# B&R Automation Studio project EFI (part 15)

#### Motors.st
```iecst
ACTION dataToMotors:
	rJogSpeedSetPoint:=data.parameters.JogSpeed;

	//Drive Unit data Managment
	MotorDriveUnit.TransmissionData := data.parameters.DriveUnit;

	MotorDriveUnit.HomePositionDesired:=data.Motor[iIndexIclaMotor].rHomePosition;;
	MotorDriveUnit.Calculation:=CALC_HOMEPOS_PULSES;
	MotorDriveUnit();

	MotorDriveUnit.SpeedDesired:=data.parameters.Speed;
	MotorDriveUnit.Calculation:=CALC_SPEED_PULSES;
	MotorDriveUnit();

	MotorDriveUnit.JogSpeedDesired:=rJogSpeedSetPoint;
	MotorDriveUnit.Calculation:=CALC_JOGSPEED_PULSES;
	MotorDriveUnit();

	MotorDriveUnit.AccelerationDesired:=data.parameters.Acceleration;
	MotorDriveUnit.Calculation:=CALC_ACC_PULSES;
	MotorDriveUnit();

	AssignDataToMotors;
END_ACTION

ACTION AssignDataToMotors:

	//Position
	//IclaMotors[iIndexIclaMotor].Parameter.MoveAbsolute.Position := REAL_TO_DINT(MotorDriveUnit.pulsesPositionDesired);

	//Speed
	IclaMotors[iIndexIclaMotor].Parameter.MoveAbsolute.Velocity := REAL_TO_UINT(MotorDriveUnit.pulsesSpeedDesired);

	//Jog Speed
	IclaMotors[iIndexIclaMotor].Parameter.Jog.VeloSlow 			:= REAL_TO_UINT(MotorDriveUnit.pulsesJogSpeedDesired);
	IclaMotors[iIndexIclaMotor].Command.JogFastSpeed 			:= FALSE;

	//Acceleration
	IclaMotors[iIndexIclaMotor].Parameter.iAcceleration 		:= REAL_TO_UINT(MotorDriveUnit.pulsesAccelerationDesired);

	//Home
	IclaMotors[iIndexIclaMotor].Parameter.Home.Position 		:= REAL_TO_DINT(MotorDriveUnit.pulsesHomePositionDesired);

	//Reset
	IclaMotors[iIndexIclaMotor].Command.Reset 					:= 	data.commands.xResetMotor OR (data.commands.xErrorRst AND
																	IclaMotors[iIndexIclaMotor].Status.IclaStatus <> AXISILE_MOVE_ABSOLUTE AND
																	IclaMotors[iIndexIclaMotor].Status.IclaStatus <> AXISILE_JOG AND
																	IclaMotors[iIndexIclaMotor].Status.IclaStatus <> AXISILE_HOMING);

END_ACTION

ACTION dataFromMotors:

	xAnyManualMovement:= (IclaMotors[iIndexIclaMotor].Status.IclaStatus = AXISILE_JOG);

	MotorDriveUnit.pulsesDevice 	:= DINT_TO_REAL(IclaMotors[iIndexIclaMotor].Status.iActualPosition);
	MotorDriveUnit.PulsesSpeedDevice:=IclaMotors[iIndexIclaMotor].Status.iActualVelocity;

	// Conversions
	MotorDriveUnit.Calculation:= CALC_POS_MM;
	MotorDriveUnit();
	rPositionMotorMm := data.Motor[iIndexIclaMotor].iDirection * MotorDriveUnit.PositionDevice;

	data.Motor[iIndexIclaMotor].rPositionMotor := rPositionMotorMm;
	data.Motor[iIndexIclaMotor].rMetalStrapPos := ABS(rPositionMotorMm)*2 + gEdgeHoldDown.Hw.rMinWidthAdjustment;

	MotorDriveUnit.Calculation:= CALC_SPEED_MM;
	MotorDriveUnit();

END_ACTION
```

- Program Logical/ExtPack/_Transport/PairedIclaMotors/PairedIclaMotorsSim/PairedIclaMotorsSim_v1/PairedIclaMotorsSim (IEC) (no source held here)

### Program Logical/ExtPack/_Transport/PairedIclaMotors/PairedIclaMotorsSim/PairedIclaMotorsSim_v1/InitPairedIclaMotorsSim (IEC)

#### InitPairedIclaMotorsSim.st
```iecst
PROGRAM _CYCLIC
	iPairedIclaMotorSimIndex := 1;
END_PROGRAM
```

### Program Logical/ExtPack/_Transport/TransVacuumCtrl/TransVacuumCtrl_v1/TransVacuumCtrl (IEC)

#### TransVacuumCtrl.var
```iecst
VAR
	dataVacc : REFERENCE TO TransVacuum_typ;
	AlarmsSummaryReseted : stEFI_AlarmSummary;
	AlarmsReseted : TransVacuumAlarms_typ;
	CommandsReseted : TransVacuumCommands_typ;
	Blower : REFERENCE TO AxisP66_typ;
	BlowersWatch : ARRAY[1..MAX_LAST_MOTOR_BLOWER] OF AxisP66_typ;
	ConditionStart_copy : BOOL; (*Storing all previous data*)
	ConditionStart : BOOL; (*Storing all previous data*)
	ConditionsStart_copy : ARRAY[1..MAX_LAST_MOTOR_BLOWER] OF BOOL; (*Storing all previous data*)
	rVacPressure : REAL; (*Pressure measured by the sensor*)
	rVacPressurePerc : REAL; (*Pressure measured by the sensor in % of MaxSystemVacuum*)
	xEnablePID : BOOL;
	xUpdatePID : BOOL;
	fbPIDPressure : MTBasicsPID;
	pidParPressure : MTPIDParametersType;
	StatusCtrl : TransVacuumStatusCtrl;
	xRunBlowerAuto : BOOL;
	xRunOutOfProduction : BOOL;
	xRunBlowerMan : BOOL;
	iReasonStop : UDINT;
	iReasonCritical : UDINT;
	iReasonSound : UDINT;
	arxAlrVacuumSensor : AutoResetSound;
	arxAlrComsBlower : AutoResetSound;
	arxAlrDriveBlowerError : AutoResetSound;
	stEventLog : EventLog_typ;
	tonJunctionAlarm : TON;
	arxAlrJointSystemPressure : AutoResetSound;
	arxAlrBlowerCB : AutoResetSound;
	uiIndex : USINT;
	StatusCtrl_copy : TransVacuumStatusCtrl;
	FLP_PresFilterPasLow : MTFilterLowPass;
	TON_StopBlowersDly : TON; (*Delay to filter fast pause-start transcition*)
	xLabStartedBlowers : BOOL; (*Blowers started for first time un the laboratory mode*)
	xAllBlowersAtSpeed : BOOL;
	xAllBlowersRunning : BOOL;
	BlowerDirection : MotorDirection_enum;
	BlowerDirectionsWatch : ARRAY[1..MAX_LAST_MOTOR_BLOWER] OF MotorDirection_enum;
	tonBlowerNotRunning : ARRAY[1..MAX_LAST_MOTOR_BLOWER] OF TON;
	iReasonOutOfProduction : UINT;
	iReasonRunAuto : USINT;
	xDisableBlower : ARRAY[1..MAX_LAST_MOTOR_BLOWER] OF BOOL;
	xAllBlowerDisabled : BOOL;
	tonBlowersRunning : TON;
	xProductionOrJamRecovery : BOOL;
	tpEvEvacuateInk : TP;
	tofNotStartAfterEStop : TOF;
	iAnyWarning : USINT;
	tonCheckAlarms : TON;
	xEnteringPowerOn : BOOL;
END_VAR
```

#### Alarms.st
```iecst
ACTION Alarms:

	IF dataVacc.Inputs.xPressureSensorError AND (xProductionOrJamRecovery OR xRunOutOfProduction) THEN
		dataVacc.Alarms.xAlrVacuumSensor := TRUE;
	END_IF

	IF dataVacc.Parameters.Hw.xSystemWithJoints THEN
		tonJunctionAlarm.IN:= NOT dataVacc.Inputs.xJointSystemPressure AND StatusCtrl<>TRANSVAC_OFF;
		tonJunctionAlarm.PT:= T#500ms;
		tonJunctionAlarm();
	END_IF

	IF tonJunctionAlarm.Q  THEN
		dataVacc.Alarms.xAlrJointSystemPressure := TRUE;
	END_IF

	IF dataVacc.Inputs.xBlowersAnyCB THEN
		dataVacc.Alarms.xAlrBlowersAnyCB := TRUE;
	END_IF

	//////////////////////////////////////////////////////////////
	// ALARMS SUMMARY    ALARMS SUMMARY    ALARMS SUMMARY

	iReasonStop.0 := dataVacc.Alarms.xAlrVacuumSensor; //To enable go to ByPass with a sensor error
	iReasonStop.1 := dataVacc.Alarms.xAlrComsBlower;
	iReasonStop.2 := dataVacc.Alarms.xAlrDriveBlowerError;
	iReasonStop.3 := dataVacc.Alarms.xAlrOvertorque;
	iReasonStop.4 := dataVacc.Alarms.xAlrJointSystemPressure AND NOT dataVacc.Parameters.AutoMode.xBypass;
	iReasonStop.5 := dataVacc.Alarms.xAlrBlowersAnyCB;
	iReasonStop.6 := dataVacc.Alarms.xAlrBlowerCB[1];
	iReasonStop.7 := dataVacc.Alarms.xAlrBlowerCB[2];
	iReasonStop.8 := dataVacc.Alarms.xAlrBlowerNotRunning[1];
	iReasonStop.9 := dataVacc.Alarms.xAlrBlowerNotRunning[2];

	IF (dataVacc.Parameters.AutoMode.xProduction OR (dataVacc.parSw.xActiveOutOfProduction AND (dataVacc.Parameters.AutoMode.xLaboratory OR dataVacc.Parameters.AutoMode.xBypass))) THEN
		dataVacc.AlSummary.xAlarmStop:=	iReasonStop > 0;
		IF EDGEPOS(dataVacc.AlSummary.xAlarmStop) THEN
			dataVacc.AlSummary.iReasonStop[0] := iReasonStop;
			LogStopAlarm;
		ELSIF EDGEPOS(NOT dataVacc.Parameters.AutoMode.xStop AND NOT dataVacc.AlSummary.xAlarmStop) THEN
			dataVacc.AlSummary.iReasonStop[0] := 0;
		END_IF
	END_IF

	dataVacc.AlSummary.xAlarmCritical := iReasonCritical > 0;
	IF EDGEPOS(dataVacc.AlSummary.xAlarmCritical) THEN
		dataVacc.AlSummary.iReasonCritical := iReasonCritical;
	ELSIF EDGEPOS(dataVacc.Parameters.Mode.xAuto AND NOT dataVacc.AlSummary.xAlarmCritical) THEN
		dataVacc.AlSummary.iReasonCritical := 0;
	END_IF

	//Warning
	// It is just used for drive alarms
	iAnyWarning.0 := dataVacc.Alarms.xAlrBlowerNotRunning[1];
	iAnyWarning.1 := dataVacc.Alarms.xAlrBlowerNotRunning[2];
	dataVacc.AlSummary.xAnyWarning:= iAnyWarning > 0;

	IF EDGEPOS(dataVacc.AlSummary.xAnyWarning) THEN
		dataVacc.AlSummary.iReasonWarning := iAnyWarning;
		//LogWarningAlarm;
	ELSIF EDGENEG(dataVacc.AlSummary.xAnyWarning) THEN
		dataVacc.AlSummary.iReasonWarning := 0;
	END_IF

	// Reseteable alarms
	arxAlrVacuumSensor.xAlarm   := dataVacc.Alarms.xAlrVacuumSensor;
	arxAlrVacuumSensor.xSilence := dataVacc.Commands.xMute;
	arxAlrVacuumSensor();

	arxAlrComsBlower.xAlarm   := dataVacc.Alarms.xAlrComsBlower;
	arxAlrComsBlower.xSilence := dataVacc.Commands.xMute;
	arxAlrComsBlower();

	arxAlrDriveBlowerError.xAlarm   := dataVacc.Alarms.xAlrDriveBlowerError;
	arxAlrDriveBlowerError.xSilence := dataVacc.Commands.xMute;
	arxAlrDriveBlowerError();

	arxAlrJointSystemPressure.xAlarm   := dataVacc.Alarms.xAlrJointSystemPressure;
	arxAlrJointSystemPressure.xSilence := dataVacc.Commands.xMute;
	arxAlrJointSystemPressure();

	arxAlrBlowerCB.xAlarm	:=	dataVacc.Alarms.xAlrBlowersAnyCB OR
								dataVacc.Alarms.xAlrBlowerCB[1] OR
								dataVacc.Alarms.xAlrBlowerCB[2];

	arxAlrBlowerCB.xSilence	:= dataVacc.Commands.xMute;
	arxAlrBlowerCB();

	iReasonSound.0 := arxAlrVacuumSensor.xAlarmSound;
	iReasonSound.1 := arxAlrComsBlower.xAlarmSound;
	iReasonSound.2 := arxAlrDriveBlowerError.xAlarmSound;
	iReasonSound.3 := arxAlrJointSystemPressure.xAlarmSound;
	iReasonSound.4 := arxAlrBlowerCB.xAlarmSound;
	dataVacc.AlSummary.xAlarmSound:= iReasonSound > 0;

	// Mute sound in belt alarms
	IF dataVacc.Commands.xMute OR dataVacc.Commands.xReset THEN
		dataVacc.AlSummary.xAlarmSound:= FALSE;
	END_IF

END_ACTION

ACTION ResetAlarms:
	dataVacc.Alarms := AlarmsReseted;
	dataVacc.AlSummary := AlarmsSummaryReseted;
END_ACTION
```

### TransVacuumSim.var
```iecst
VAR
	iTransVacummSimIndex : USINT;
END_VAR
```

### Program Logical/ExtPack/_Transport/TransVacuumCtrl/TransVacuumSim/TransVacuumSim_v1/InitTransVacuumSim

#### Cyclic.st
```iecst
PROGRAM _CYCLIC
	(* Insert code here *)
	iTransVacummSimIndex := 1;

END_PROGRAM
```

### Program Logical/ExtPack/_Transport/TransVacuumCtrl/TransVacuumSim/TransVacuumSim_v1/TransVacuumSim (IEC)

#### TransVacuumSim.var - Local variables
```iecst
VAR
	transVacc : REFERENCE TO TransVacuum_typ;
	pressureSim : SimAnalogProcess;
	rAParam : REAL := -0.13;
	rBParam : REAL := -0.005;
	tofNoVacc : TOF;
END_VAR
```

### Program Logical/ExtPack/BlockCtrl/BlockCtrl_v1/BlockCtrl (IEC) - Block program

#### BlockParameters.st
```iecst
ACTION BlockParameters:

	//Cleaning offset limits.(antes en securities)
	Block.parSw.rOffsetCleanMtrAdjust	:= LIMIT(Block.parameters.Motor.rMinCleanOffsetTech, Block.parSw.rOffsetCleanMtrAdjust, Block.parameters.Motor.rMaxCleanOffsetTech);
	Block.parSw.rOffsetCleanMtrOperatr := LIMIT(-1, Block.parSw.rOffsetCleanMtrOperatr, 1);

	// Clean offset
	rOffseCleanMtr:=Block.parSw.rOffsetCleanMtrAdjust+Block.parSw.rOffsetCleanMtrOperatr;

	//Minimum position of the Motor to allow moving the Icla in Manual mode
	rSafeBarPosToCarrier := Block.parameters.Motor.rSafePositionCleanCarrier; //Block.parameters.Motor.rCleanPosition + rOffseCleanMtr;

	// rWaterSpurtPosition always has to be higher than rCleanPosition
	IF Block.parameters.Motor.rWaterSpurtPosition <= Block.parameters.Motor.rCleanPosition + 0.5 THEN
		Block.parameters.Motor.rWaterSpurtPosition := Block.parameters.Motor.rCleanPosition + 0.5;
	END_IF

	// Print motor offset
	IF NOT Block.parameters.xMotorOffsetAllowed THEN
		Block.parSw.rOffsetPrintMotor := 0;
	ELSE
		Block.parSw.rOffsetPrintMotor := MAX(Block.parSw.rOffsetPrintMotor,GC_MIN_OFFSET_BLOCK);
	END_IF

	// Clean motor speed limits
	Block.parameters.Icla.iCleanMotorSpeedFwd:= LIMIT(Block.parameters.Icla.iMinSpeedCleanMotorFwd,
														Block.parameters.Icla.iCleanMotorSpeedFwd,
														Block.parameters.Icla.iMaxSpeedCleanMotorFwd);

	Block.parameters.Icla.iCleanMotorSpeedBwd:= LIMIT(Block.parameters.Icla.iMinSpeedCleanMotorBwd,
														Block.parameters.Icla.iCleanMotorSpeedBwd,
														Block.parameters.Icla.iMaxSpeedCleanMotorBwd);

	//Assign the direction of the vertical motor
	IF Block.parameters.Motor.VerticalDirection=MOTOR_NEGATIVE THEN
		AxisBK.Parameter.Direction:=MOTOR_NEGATIVE_AXIS;
	ELSE
		AxisBK.Parameter.Direction:=MOTOR_POSITIVE_AXIS;
	END_IF

	Block.parameters.Inks.iMaxMachinePrintBars := MIN(Block.parameters.Inks.iMaxMachinePrintBars, MAX_LAST_INK);

END_ACTION
```

#### AlarmSound.st - Assign sound to alarms
```iecst
ACTION AlarmSound:

	//////////////////////////////
	// BLOCK SOUNDS
	//////////////////////////////

	// Block sounds while is homing
	// Sound generation for homing process
	// Sound generation: manual movements
	xAnyManualMov	:=	Block.Status.Motor.xBarsHoming OR
						AxisBK.Command.Jog.ContinuousPos OR
						AxisBK.Command.Jog.ContinuousNeg OR
						IclaBK.Command.JogForward OR
						IclaBK.Command.JogBackward;

	// Reseteable alarms. Reset is input in the ars function
	// Alarms reseteable sound management.
	ars_AlrStop.xAlarm:= Block.AlSummary.xAlarmStop;
	ars_AlrStop.xSilence:= Block.commands.xMute;
	ars_AlrStop();

	ars_AlrCritical.xAlarm:= Block.AlSummary.xAlarmCritical;
	ars_AlrCritical.xSilence:= Block.commands.xMute;
	ars_AlrCritical();

	ars_AlrWarning.xAlarm:= Block.AlSummary.xAnyWarning;
	ars_AlrWarning.xSilence:= Block.commands.xMute;
	ars_AlrWarning();

	//reasonSound.0 := ars_AlrWarning.xAlarmSound;  //[RGP] I think warnings shouldnt sound
	reasonSound.1 := ars_AlrStop.xAlarmSound;
	reasonSound.2 := ars_AlrCritical.xAlarmSound;
	reasonSound.3 := (xAnyManualMov AND gPLC.xBlk_200ms);

	Block.AlSummary.xAlarmSound := reasonSound>0;

END_ACTION
```

#### AlarmsSummary.st - Alarms summary
```iecst
ACTION AlarmsSummary:

	// Stop Alarms. The machine goes to Automatic-Stop.
	iReasonStop.0 := Block.Al.xAlrCleanMtrNoRef;
	iReasonStop.1 := Block.Al.xAlAirVenturi AND Block.Status.PositionState = BLOCKP_CLEANING;
	iReasonStop.2 := Block.Al.xAnyVerticalDriveAlarm;
	iReasonStop.3 := Block.Al.xAlrBarMtrNoRef;
	iReasonStop.4 := Block.Al.xSiUnitPowerOff;
	iReasonStop.5 := Block.Al.xAlrComSiUnit;
	iReasonStop.6 := Block.Al.xAlrComBarMtr;
	iReasonStop.7 := Block.Al.xAlrCleanMotor;
	iReasonStop.8 := Block.Al.xAlrComCleanMtr;
	iReasonStop.9 := Block.Al.xAlrEnabCleanMtrDiffLvL;
	iReasonStop.10 := Block.Al.xAlrIncoherPositCleanMtr;
	iReasonStop.11 := Block.Al.xAlCleanInterrupt AND Block.commands.AutoMode.xProdORLab;
	iReasonStop.12 := (Block.Al.xAlrTraySensor OR Block.Al.xAlrCleanSensor) AND Block.commands.AutoMode.xProdORLab;
	iReasonStop.13 := Block.Al.xNoActionDangerCollision;
	iReasonStop.14 := Block.Al.xAlrControllerNotReady;
	iReasonStop.15 := Block.Al.xAlrOverTorque;

	Block.AlSummary.xAlarmStop:= iReasonStop > 0;
	IF EDGEPOS(Block.AlSummary.xAlarmStop) THEN
		Block.AlSummary.iReasonStop[0] := iReasonStop;
		LogStopAlarm;
	ELSIF EDGEPOS(NOT Block.commands.AutoMode.xStop AND NOT Block.AlSummary.xAlarmStop) THEN
		Block.AlSummary.iReasonStop[0] := 0;
	END_IF

	// Out of Automatic Alarms. The machine goes to Standby mode.
	iReasonCritical.0 := (Block.Al.xAlrSafetySystemInBlock AND Block.Status.xEnabledMovements);
	iReasonCritical.1 := Block.Al.xAlrDif;
	iReasonCritical.2 := Block.Al.xAlrDriveProtection;
	Block.AlSummary.xAlarmCritical:= iReasonCritical > 0;

	//Register the reason of the Critical Alarm
	IF Block.commands.Mode.xAuto AND EDGEPOS(Block.AlSummary.xAlarmCritical) THEN
		Block.AlSummary.iReasonCritical := iReasonCritical;
		LogCriticalAlarm;
	ELSIF EDGEPOS(Block.commands.Mode.xAuto AND NOT Block.AlSummary.xAlarmCritical) THEN
		Block.AlSummary.iReasonCritical := 0;
	END_IF

	// Any alarm
	Block.AlSummary.xAnyAlarm:= Block.AlSummary.xAlarmStop OR Block.AlSummary.xAlarmCritical;

	// Warning alarms (used in AlarmaAvisoExterno)
	iReasonAnyWarning.0 := Block.Al.xAlrNoTrayInServoNoHomed;
	iReasonAnyWarning.1 := Block.Al.xModuleTemp01;
	iReasonAnyWarning.2 := Block.Al.xModuleTemp02;
	iReasonAnyWarning.3 := Block.Al.xModuleTemp03;
	iReasonAnyWarning.4 := Block.Al.xModuleTemp04;
	iReasonAnyWarning.5 := Block.Al.xBarDriverTemp;
	iReasonAnyWarning.6 := Block.Al.xBarMotorTemp;
	iReasonAnyWarning.7 := Block.Al.xAlrCheckHomingSensor;
	iReasonAnyWarning.8 := Block.Al.xAlrBlockReachedMaxPosition;
	iReasonAnyWarning.9 := Block.Al.xAlrTempPowerSupply;
	iReasonAnyWarning.10 := Block.Al.xAlrDecreaseCleanOffset;
	iReasonAnyWarning.11 := Block.Al.xAlrCappingWaterTankEmpty;
	iReasonAnyWarning.12 := Block.Al.xAlrCappingWaterNotRecirc;
	iReasonAnyWarning.13 := Block.Al.xAlrReferenceIncoherence;
	iReasonAnyWarning.14 := Block.Al.xAlrWtrPresSensBroken;
	iReasonAnyWarning.15 := Block.Al.xAlrWaterPumpPresure;
	iReasonAnyWarning.16 := Block.Al.xAlrEmptyWaterTank;
	iReasonAnyWarning.17 := Block.Al.xWrnOverTorq;

	Block.AlSummary.xAnyWarning:= iReasonAnyWarning > 0 ;

	//Alarm Safety System General
	iReasonSafetyGeneral.1 := Block.Al.xAlrSafetySystemInBlock;
	iReasonSafetyGeneral.2 := Block.Al.xAlrFrontEmergencyStop;
	iReasonSafetyGeneral.3 := Block.Al.xAlrRearEmergencyStop;
	iReasonSafetyGeneral.4 := Block.Al.xAlrLogicEmergencyStop;
	iReasonSafetyGeneral.5 := xAnyUpperSafety AND Block.commands.AutoMode.xProdORLab;
	iReasonSafetyGeneral.6 := NOT Block.In.Safety.xSafetyOK;
	Block.AlSummary.xAlrSafetySystemGeneral:= iReasonSafetyGeneral > 0;

	iReasonSafetyCutAir.0 := Block.Al.xAlrSafetySystemInBlock;
	iReasonSafetyCutAir.1 := Block.Al.xAlrFrontEmergencyStop;
	iReasonSafetyCutAir.2 := Block.Al.xAlrRearEmergencyStop;
	iReasonSafetyCutAir.3 := Block.Al.xAlrLogicEmergencyStop;
	iReasonSafetyCutAir.4 := xAnyUpperSafety;
	Block.AlSummary.xAlrSafetyCutAir:= iReasonSafetyCutAir > 0;

END_ACTION
```

#### ResetAlarms.st - Reset alarms
```iecst
ACTION ResetAlarms:

	Block.Al:= stBlockAlarmsReseted;
	Block.AlSummary:= stBlockAlarmsSummaryReseted;
	xCleanInterrupt:=FALSE;

END_ACTION
```

#### ControlState.st - Block states
```iecst
ACTION ControlState:

	// General states
	Block.Status.Motor.xBarsHoming:= AxisBK.Status.PLCopenState.Homing; //  States for Homing block
	Block.Status.Motor.ErrorID := AxisBK.Status.ErrorID;
	Block.Status.Motor.ActPosition := REAL_TO_UDINT(AxisBK.Status.ActPosition);

	//Motor status read from drives
	//Torque
	Block.Status.Motor.rActTorque	:= ABS(AxisBK.Status.ActTorque);
	Block.Status.Motor.rMaxTorque	:= ABS(AxisBK.Status.MaxTorque);
	Block.Status.Motor.rRatedTorque	:= ABS(AxisBK.Status.RatedTorque);

	IF NOT Block.parameters.Motor.xOversized THEN
		Block.Status.Motor.rOperationTorque := Block.Status.Motor.rRatedTorque;
	ELSE
		Block.Status.Motor.rOperationTorque := Block.parameters.Motor.rOperationTorque;
	END_IF

	//Temp
	Block.Status.Motor.rActTemp	:= AxisBK.Status.ActTempMot;
	Block.Status.Motor.rMaxTemp	:= AxisBK.Status.MaxTempMotor;
	Block.Status.Motor.rSpeed	:= AxisBK.Status.ActVelocity;

	//Velocity
	MotorDriveUnit.PulsesSpeedDevice := AxisBK.Status.ActVelocity;
	MotorDriveUnit.Calculation := CALC_SPEED_MM;
	MotorDriveUnit();
	Block.Status.Motor.rActVelocity := MotorDriveUnit.SpeedDevice;

	MotorDriveUnit.PulsesSpeedDevice := AxisBK.Status.MaxSpeed;
	MotorDriveUnit.Calculation := CALC_SPEED_MM;
	MotorDriveUnit();
	Block.Status.Motor.rMaxVelocity := MotorDriveUnit.SpeedDevice;

	//Icla
	Block.Status.Icla.xHomed:= Block.Status.Icla.xHomed;
	Block.Status.Icla.xHoming := Block.Status.PositionState = BLOCKP_HOMING_ICLA; //Those are the states for Homing
	Block.Status.Icla.ErrorNumber:=IclaBK.Status.Error.ErrorNumber;
	Block.Status.Icla.xInError := IclaBK.Status.xInError;

	//Torque
//	Block.Status.Icla.rActTorque	:= IclaBK.Status.iActualVelocity;
//	Block.Status.Icla.rMaxTorque	:= IclaBK.Status.iActualVelocity;

	//Temp
//	Block.Status.Icla.rActTemp	:= IclaBK.Status.iActualVelocity;
//	Block.Status.Icla.rMaxTemp	:= IclaBK.Status.iActualVelocity;

	//Velocity
	Block.Status.Icla.iSpeed := IclaBK.Status.iActualVelocity;
//	Block.Status.Icla.iMaxSpeed := IclaBK.Status.iActualVelocity;

	xAnyManualMovement:=(AxisBK.Status.PLCopenState.ContinuousMotion OR xIclaMoving OR Block.Status.Icla.xHoming) AND (Block.commands.Mode.xManual);
	Block.Status.xAnyManualMovement:=xAnyManualMovement;

END_ACTION
```

#### BlockStatesCtrl.st - State machine ctrl block states
```iecst
ACTION BlockStatesCtrl:

	//Desired print position is max value because rPrintPosition comes form belt algorithm corecction based on matrix at LC_Band.st. It gives rPrintPosition calculated by matrix
	IF Block.commands.StateMode = PRINTERGEN_AUTO THEN
		rCalcPosDesPrint:= MAX (Block.parameters.Motor.rPrintPosition + Block.parSw.rOffsetPrintMotor,
							Block.parameters.Motor.rMinSafePosition + Block.parSw.rOffsetPrintMotor);
	ELSIF (Block.commands.StateMode = PRINTERGEN_MANUAL) AND Block.commands.Manual.xToPrintPosition THEN
		rCalcPosDesPrint:= Block.parameters.rManPrintingPos;
	END_IF

	//If PreprintingPosition is forced, recalculate the desired position
	IF Block.commands.xForcePreprintingPos THEN
		rCalcPosDesPrint:= MAX (rCalcPosDesPrint, Block.parameters.rPrePrintingPos);
	END_IF

	//Manage Block.Status.BlockState depending on the MachineMode
	//	PRINTERGEN_ZERO:
	//	PRINTERGEN_MANUAL:
	//	PRINTERGEN_AUTO:
	BlockStateMach;

	//Manage the General State of the BLOCK
	//	BLOCK_STOPPED:
	//	BLOCK_STOPPING:
	//	BLOCK_MANUAL:
	//	BLOCK_AUTO:
	BlockStateGen;

	//Manage the current position of the Block
	//	BLOCKP_UNDEFINED:
	//	BLOCKP_HOMING_ICLA:
	//	BLOCKP_HOMING_BAR:
	//	BLOCKP_IN_CAP:
	//	BLOCKP_IN_PRINT:
	//	BLOCKP_IN_CLEAN:
	//	BLOCKP_CLEANING:
	//	BLOCKP_GOING_TO_CAP:
	//	BLOCKP_GOING_TO_PRINT:
	//	BLOCKP_GOING_TO_CLEAN:
	PreviousLogic;
	BlockStatePos;
	PosteriorLogic;

	LogOrders;
	DefineBoolPositionStatus;
	RegisterCyclesInPosState;

	BlockStatePrevious := Block.Status.BlockState;
	MachineStatePrevious :=  Block.commands.StateMode;

END_ACTION

ACTION StopMovements:

	Block.Out.xTrayOut:=FALSE;
	Block.Out.xTrayIn:=FALSE;
	Block.Out.xVenturi:=FALSE;
	Block.Out.xCleaningWaterPump:=FALSE;
	Block.Out.xCappingWaterPump:=FALSE;
	Block.Out.xWastedInkTankPump:=FALSE;

	StopBar;
	StopIcla;

END_ACTION

ACTION RegisterCyclesInPosState:

	//BlockStates to SW and times in each position
	CASE Block.Status.PositionState OF
		BLOCKP_UNDEFINED:		Block.Status.iBlockState:= 0; iTimesStateBlockUndefined := iTimesStateBlockUndefined+1;
		BLOCKP_HOMING_BAR:		Block.Status.iBlockState:= 0; iTimesStateBlockHomingBar := iTimesStateBlockHomingBar+1;
		BLOCKP_HOMING_ICLA:		Block.Status.iBlockState:= 0; iTimesStateBlockHomingIcla := iTimesStateBlockHomingIcla+1;
		BLOCKP_IN_CAP:			Block.Status.iBlockState:= 1; iTimesStateBlockInCap := iTimesStateBlockInCap+1;
		BLOCKP_IN_PRINT:		Block.Status.iBlockState:= 2; iTimesStateBlockPrinting := iTimesStateBlockPrinting+1;
		BLOCKP_CLEANING:		Block.Status.iBlockState:= 3; iTimesStateBlockCleaning := iTimesStateBlockCleaning+1;
		BLOCKP_GOING_TO_CAP:	Block.Status.iBlockState:= 4; iTimesStateBlockGoingToCap := iTimesStateBlockGoingToCap+1;
		BLOCKP_GOING_TO_PRINT:	Block.Status.iBlockState:= 5; iTimesStateBlockGoingToPrint := iTimesStateBlockGoingToPrint+1;
	END_CASE

END_ACTION

ACTION DefineBoolPositionStatus:

	Block.Status.Position.xUndefined	:= 	Block.Status.PositionState = BLOCKP_UNDEFINED;
	Block.Status.Position.xInCap    	:=	Block.Status.PositionState = BLOCKP_IN_CAP;
	Block.Status.Position.xInPrint 		:=	Block.Status.PositionState = BLOCKP_IN_PRINT;
	Block.Status.Position.xInClean 		:=	Block.Status.PositionState = BLOCKP_IN_CLEAN;
	Block.Status.Position.xCleaning 	:= 	Block.Status.PositionState = BLOCKP_CLEANING;
	Block.Status.Position.xGoingToCap	:=	Block.Status.PositionState = BLOCKP_GOING_TO_CAP;
	Block.Status.Position.xGoingToPrint :=	Block.Status.PositionState = BLOCKP_GOING_TO_PRINT;
	Block.Status.Position.xGoingToClean :=	Block.Status.PositionState = BLOCKP_GOING_TO_CLEAN;

END_ACTION

ACTION ResetKnownPositions:

	xInCap:= FALSE;
	xInPrint:= FALSE;
	xInClean:= FALSE;

END_ACTION

ACTION LogOrders:

	IF  Block.Status.PositionState = BLOCKP_GOING_TO_CAP AND BlockPositionPrevious <> BLOCKP_GOING_TO_CAP THEN
		LogToCapOrder;
	END_IF
	IF Block.Status.PositionState = BLOCKP_GOING_TO_PRINT AND BlockPositionPrevious <> BLOCKP_GOING_TO_PRINT THEN
		LogToPrintOrder;
	END_IF
	IF Block.Status.PositionState = BLOCKP_CLEANING AND BlockPositionPrevious <> BLOCKP_CLEANING THEN
		LogToCleanOrder;
	END_IF

END_ACTION
```

#### BlockStateMach.st
```iecst
ACTION BlockStateMach:

	CASE Block.commands.StateMode OF

		PRINTERGEN_ZERO:
			//When entering in Zero, go to Stopping
			IF MachineStatePrevious<>PRINTERGEN_ZERO THEN
				Block.Status.BlockState := BLOCK_STOPPING;

				//Reset cleaning order and status if going to 0 while cleaning
				IF Block.Status.PositionState = BLOCKP_CLEANING THEN
					ResetCleanCycle;
				END_IF

				//If the block is not in a clear position, go to undefined
				IF Block.Status.PositionState <> BLOCKP_IN_CAP AND Block.Status.PositionState <> BLOCKP_IN_PRINT THEN
					Block.Status.PositionState := BLOCKP_UNDEFINED;
				END_IF
				nState :=0;
			END_IF

		PRINTERGEN_STARTUP:
			IF Block.Status.BlockState = BLOCK_STOPPED AND NOT Block.Status.Motor.xBarsHomed THEN
				Block.Status.BlockState := BLOCK_MANUAL;
			END_IF
			IF Block.Status.Motor.xBarsHomed THEN
				Block.Status.BlockState := BLOCK_AUTO;
			END_IF

		PRINTERGEN_MANUAL:
			IF Block.Status.BlockState = BLOCK_STOPPED THEN
				Block.Status.BlockState := BLOCK_MANUAL;
			END_IF

		PRINTERGEN_AUTO:

			IF Block.Status.BlockState = BLOCK_STOPPED AND AllDevicedHomed(ADR(Block)) THEN
				Block.Status.BlockState := BLOCK_AUTO;
			END_IF

	END_CASE

END_ACTION
```

#### BlockStatePos.st
```iecst
ACTION BlockStatePos:

	// If not in AUTO or MANUAL, no action in this section
	IF Block.Status.BlockState <> BLOCK_MANUAL AND Block.Status.BlockState <> BLOCK_AUTO THEN
		BlockPositionPrevious := BLOCKP_UNDEFINED;
		//These actions were executed originally in "BLOCKP_HOMING_BAR" and "BLOCKP_HOMING_ICLA" states respectively.
		//One of the conditions to execute it was to be in zero state, but the CASE below is not executed when in zero state
		//so adding these actions here before the RETURN
		ResetHomingBar;
		ResetHomingIcla;
		RETURN;
	END_IF

	xBlockPosChange := BlockPositionPrevious <> Block.Status.PositionState;
	BlockPositionPrevious := Block.Status.PositionState;

	CASE Block.Status.PositionState OF
		BLOCKP_UNDEFINED:
			ResetKnownPositions;
			AxisBK.Command.QuickStop := FALSE;

		BLOCKP_HOMING_ICLA:

			//Aborting Icla homing process
			IF (EDGEPOS(Block.commands.xIclaHomeOrderInterrupt) OR Block.commands.Mode.xZero OR IclaBK.Status.xInError) THEN // When printerr is St zero
				ResetHomingIcla;
				Block.Status.PositionState := BLOCKP_UNDEFINED;
			END_IF

			HomingIcla;
			IF Block.Status.Icla.xHomed THEN
				Block.Status.PositionState := BLOCKP_UNDEFINED;
			END_IF

		BLOCKP_HOMING_BAR:

			//Aborting Block Motor homing process
			iCancelHomingBar.0 := NOT Block.In.xIclaSensor OR NOT Block.In.xTrayOut;
			iCancelHomingBar.1 := NOT Block.In.xTrayOut;
			iCancelHomingBar.2 := Block.AlSummary.xAlarmCritical;
			iCancelHomingBar.3 := Block.commands.Mode.xZero;
			iCancelHomingBar.4 := NOT Block.commands.xBarHomeOrder;
			IF iCancelHomingBar > 0 THEN
				ResetHomingBar;
				Block.Status.PositionState := BLOCKP_UNDEFINED;
			END_IF

			HomingBar;
			IF Block.Status.Motor.xBarsHomed THEN
				Block.Status.PositionState := BLOCKP_UNDEFINED;
			END_IF

		BLOCKP_IN_CAP:

		BLOCKP_IN_PRINT:

			//Send and adjustment in position if needed
			IF ABS(rMotorCurrentPos-rCalcPosDesPrint)>0.01 AND ABS(rMotorAbsPosDesired - rCalcPosDesPrint)>0.01 THEN
				rMotorAbsPosDesiredPrevious := rMotorAbsPosDesired;
				rMotorAbsPosDesired:= rCalcPosDesPrint;
				MoveAbsolute;
			END_IF
			Block.Status.Position.xReadyToPrint := NOT Block.commands.xForcePreprintingPos;

		BLOCKP_CLEANING:
			Cleaning;

			//Manage cancelling a cleaning
			iCancelCleaning.0 := Block.AlSummary.xAlrSafetySystemGeneral;
			iCancelCleaning.1 := Block.Al.xAlrSafetySystemInBlock;
			iCancelCleaning.2 := Block.Al.xAnyVerticalDriveAlarm;
			iCancelCleaning.3 := Block.Al.xAlrCleanMotor;
			iCancelCleaning.4 := Block.Al.xAlrTraySensor;
			iCancelCleaning.5 := Block.Al.xAlAirVenturi;
			iCancelCleaning.6 := Block.AlSummary.xAlarmStop;
			iCancelCleaning.7 := Block.AlSummary.xAnyAlarm;
			iCancelCleaning.8 := Block.Al.xAlrFrontCurtain;
			iCancelCleaning.9 := Block.Al.xAlrFrontSafety;
			iCancelCleaning.10 := Block.Al.xAlrRearSafety;
			iCancelCleaning.11 := Block.commands.xCleanStop;
			iCancelCleaning.12 := Block.Al.xNoActionDangerCollision;
			IF EDGEPOS(iCancelCleaning > 0) THEN
				iSaveReason := iCancelCleaning;
				iSaveState := nState;
				ResetCleanCycle;
				xCleanInterrupt:=TRUE;
				Block.Status.PositionState := BLOCKP_GOING_TO_CAP;
			END_IF

		BLOCKP_GOING_TO_CAP:
			GoingToCap;
			IF xInCap THEN
				Block.Status.PositionState := BLOCKP_IN_CAP;
			END_IF

		BLOCKP_GOING_TO_PRINT:
			GoingToPrint;
			IF xInPrint THEN
				Block.Status.PositionState := BLOCKP_IN_PRINT;
			END_IF

		BLOCKP_GOING_TO_CLEAN:
			GoingToClean;
			IF xInClean THEN
				Block.Status.PositionState := BLOCKP_IN_CLEAN;
			END_IF

	END_CASE

	Block.Status.Motor.rMotorAbsPosDesired := rMotorAbsPosDesired;

	//Saving state history
	IF Block.Status.PositionState<>StatePosHistory[0] THEN
		ShiftArrayForward(ADR(StatePosHistory), SIZEOF(StatePosHistory), SIZEOF(StatePosHistory[0]), 1, iHistoryLines);
		StatePosHistory[0]:=Block.Status.PositionState;
	END_IF

END_ACTION
```

#### GeneralLogic.st
```iecst
ACTION PreviousLogic:

	//With the Sensor, always remove the alarm
	IF Block.In.xIclaSensor THEN
		Block.Al.xNoActionDangerCollision:=FALSE;
	END_IF

	tonWaitingSensor.IN := nState=212 OR nState=215 OR nState=235 OR nState=269;
	tonWaitingSensor.PT := T#3s;
	tonWaitingSensor();

	IF NOT AxisBK.Status.HomeOK THEN
		Block.Status.Motor.xBarsHomed:= FALSE;
	END_IF

	// Safety Tray Out
	IF EDGEPOS(Block.In.xTrayOut AND Block.Out.xTrayOut) THEN
		Block.Out.xTrayOut:= FALSE;
	END_IF
	// Safety Tray In
	IF EDGEPOS(Block.In.xTrayIn AND Block.Out.xTrayIn) THEN
		Block.Out.xTrayIn:= FALSE;
	END_IF

	//To wait some time to empty the water tray for capping
	TON_WaitToMoveTrayOut.IN := NOT Block.Out.xCappingWaterPump AND (nState=234);
	TON_WaitToMoveTrayOut.PT := T#5S;
	TON_WaitToMoveTrayOut();

	// Capping water pump
	IF (Block.Status.PositionState <> BLOCKP_IN_CAP) THEN
		Ton_CappingPump.IN := FALSE;
	ELSIF (Block.In.xTrayIn AND Block.parameters.xCappingProcess) THEN
		Ton_CappingPump.IN := TRUE;
	END_IF
	Ton_CappingPump.PT := T#150s;
	Ton_CappingPump();
	Block.Out.xCappingWaterPump := Ton_CappingPump.IN AND NOT Ton_CappingPump.Q;

	iReasonRunWastedInkPump.0 := EDGEPOS (Block.In.xTrayIn AND Block.parameters.xWastedInkTankProcess);
	iReasonRunWastedInkPump.1 := EDGEPOS (Block.Status.xCleaningDone AND Block.parameters.xWastedInkTankProcess);

	IF iReasonRunWastedInkPump > 0 THEN
		xStartWastedInkPump := TRUE;
	END_IF

	// Wasted ink tank
	Ton_WastedInkTankPump.IN := xStartWastedInkPump;
	Ton_WastedInkTankPump.PT := T#200s;
	Ton_WastedInkTankPump();
	Block.Out.xWastedInkTankPump := xStartWastedInkPump := Ton_WastedInkTankPump.IN AND NOT Ton_WastedInkTankPump.Q;

	IF Block.Status.PositionState <> BLOCKP_IN_PRINT THEN
		Block.Status.Position.xReadyToPrint := FALSE;
	END_IF

END_ACTION

ACTION PosteriorLogic:

	//Remove the other order when receiving a pulse. https://jira.efi.com/browse/CRETALEGO-1375
	IF EDGEPOS(Block.Out.xTrayOut) THEN Block.Out.xTrayIn:= FALSE; END_IF
	IF EDGEPOS(Block.Out.xTrayIn) THEN Block.Out.xTrayOut:= FALSE; END_IF

	// Update state
	Block.Status.iBlockCaseLogicControl:=nState;
	Block.Status.Icla.iIclaState:=IclaBK.Status.iDriveStatus;

	//NOZOMITWO-1116: Block tray movements when printer key maintenance is activated
	IF Block.parameters.xPrinterKeyMaintenanceActivated THEN
		Block.commands.Manual.xManTrayIn:= FALSE; //CUBE-963. Remove order if the movement is been blocked
		Block.commands.Manual.xManTrayOut:= FALSE; //CUBE-963. Remove order if the movement is been blocked
		Block.Out.xTrayIn:= FALSE;
		Block.Out.xTrayOut:= FALSE;
	END_IF

END_ACTION
```

#### AutoLogic.st
```iecst
ACTION GoingToCap:

	IF xBlockPosChange THEN
		nState := 208;
	END_IF

	CASE nState OF

		(*STOP POSITION     --------------------------------------------------------*)
		(*STOP POSITION     --------------------------------------------------------*)
		(*STOP POSITION     --------------------------------------------------------*)

		208:
			iLastState:=nState;
			ResetKnownPositions;
			nState:= nState+1;

		209:
			iLastState:=nState;
			IF AxisBK.Status.ErrorID=0 THEN
				StopMovements;
				nState:= nState+1;
			END_IF

		210:
			iLastState:=nState;
			IF AllDevicedStopped(ADR(Block), ADR(AxisBK), ADR(IclaBK)) THEN
				IF AxisBK.Status.PowerOn  AND AxisBK.Status.PLCopenState.StandStill THEN
					nState:= nState+1;
				END_IF
			END_IF

		211:
			iLastState:=nState;

			//If It is in safe place we go to next step
			IF ABS(rMotorCurrentPos-Block.parameters.Motor.rCapPosition)<0.01 THEN
				nState:= nState+3;
				//If bars are up than tray its not necessary move tray out
			ELSIF (rMotorCurrentPos > (Block.parameters.Motor.rCappingPosition - 0.05) AND Block.parameters.xCappingProcess) OR
				(rMotorCurrentPos > (Block.parameters.Motor.rDripBarsPosition + 0.01) AND NOT Block.parameters.xCappingProcess) THEN
				MoveBarsToCapPosition;
				nState:= nState+2; //To go to CheckAbsolutMovementFinished state
			ELSE
				//Tray Out
				Block.Out.xTrayOut:= TRUE;
				nState:= nState+1;
			END_IF

		212:
			iLastState:=nState;
			//Waiting the Tray to be out and ready to move
			IF Block.In.xTrayOut THEN
				MoveBarsToCapPosition;
			END_IF

		213:
			iLastState:=nState;

			CheckAbsolutMovementFinished;

		214:// Icla Position check
			iLastState:=nState;

			//If Icla is in position, jump 2 steps
			IF Block.In.xIclaSensor  THEN
				nState:= nState+2;
			//If Icla is not in position, send the order and jump 1 step to wait the move
			ELSE
				//Cleaning Motor going to stop position
				rIclaAbsPosDesired:= Block.parameters.Icla.rPositionCleanMotorBwd;
				IclaBK.Parameter.MoveAbsolute.Velocity:= INT_TO_UINT(Block.parameters.Icla.iCleanMotorSpeedBwd);
				xIclaAbsMovOrder:=TRUE;
				nState:= nState+1;
			END_IF

		215:
			iLastState:=nState;

			IF Block.In.xIclaSensor THEN
				xIclaAbsMovOrder:=FALSE;
				nState:= nState+1;
			END_IF

		216:
			iLastState:=nState;

			//Be sure to place the tray in position
			Block.Out.xTrayIn:= TRUE;
			nState:= nState+1;

		217:
			iLastState:=nState;
			// Check that s not true other wise we tray in again
			IF NOT Block.In.xTrayOut AND Block.In.xTrayIn THEN
				IF Block.parameters.xCappingProcess AND Block.In.xFrontDoorClosed THEN
					MoveBarsToCappingPosition;
				ELSE
					nState:= nState+1;
				END_IF
			END_IF

		218:
			iLastState:=nState;
			// Check that s not true other wise we tray in again
			IF Block.parameters.xCappingProcess THEN
				CheckAbsolutMovementFinished;
			ELSE
				nState:= nState+1;
			END_IF

		219:
			iLastState:=nState;
			xInCap:= TRUE;
			nState:= 0;

	END_CASE

END_ACTION

ACTION GoingToPrint:

	IF xBlockPosChange THEN
		nState := 230;
	END_IF

	CASE nState OF

		(*PRINT POSITION    --------------------------------------------------------*)
		(*PRINT POSITION    --------------------------------------------------------*)
		(*PRINT POSITION    --------------------------------------------------------*)

		230:
			iLastState:=nState;

			ResetKnownPositions;

			nState:= nState+1;

		231:
			iLastState:=nState;
			IF AxisBK.Status.ErrorID=0 THEN
				StopMovements;
				nState:= nState+1;
			END_IF

		232:
			iLastState:=nState;
			IF AllDevicedStopped(ADR(Block), ADR(AxisBK), ADR(IclaBK)) THEN
				IF AxisBK.Status.PowerOn AND AxisBK.Status.PLCopenState.StandStill THEN
					nState:= nState+1;
				END_IF
			END_IF

		233:
			iLastState:=nState;
			// Checking icla position (Could it produce crashes?)
			IF Block.In.xIclaSensor THEN
				xIclaAbsMovOrder:= FALSE;
				IF (NOT Block.parameters.xCappingProcess) THEN
					nState:= nState+1;
				ELSE
					IF ABS(rMotorCurrentPos-Block.parameters.Motor.rCappingPosition)<0.01 THEN
						MoveBarsAboveCappingPosition;
					ELSE
						nState:= nState+1;
					END_IF
				END_IF
			END_IF

		234:
			iLastState:=nState;

			//Tray out to allow go down
			xWaitToMoveTrayOut := (TON_WaitToMoveTrayOut.Q OR NOT Block.parameters.xCappingProcess);
			IF xWaitToMoveTrayOut THEN
				IF (NOT Block.In.xTrayOut) THEN
					Block.Out.xTrayOut:= TRUE;
				END_IF
				nState:= nState+1;
			END_IF

		235:
			iLastState:=nState;
			//Tray out to allow go down
			ton_TrayOut(IN:=Block.In.xTrayOut, PT:=T#2S);
			IF ton_TrayOut.Q  THEN
				nState:= nState+1;
			END_IF

		236:
			iLastState:=nState;
			//Going to print
			MoveBarsToPrintingPosition;

		237:
			iLastState:=nState;

			IF ABS(rMotorCurrentPos-rMotorAbsPosDesired)<0.01 THEN
				xInPrint:= TRUE;
				nState:= 0;
			END_IF

	END_CASE

END_ACTION

ACTION Cleaning:

	IF xBlockPosChange THEN
		nState := 250;
	END_IF

	// Drip Control Time established by user
	TON_DRIPPING.IN:= Block.commands.xDripControl;
	TON_DRIPPING.PT:= tiDripTimeMax;
	TON_DRIPPING ();
	xFinishedDrippingOrderByBlock:=TON_DRIPPING.Q;
	IF xFinishedDrippingOrderByBlock THEN
		Block.commands.xDripControl:= FALSE;
	END_IF

	//Delay after Drip state
	tonStabInksAfterDrip.IN:=(nState=258);
	tonStabInksAfterDrip.PT:=T#3S;
	tonStabInksAfterDrip();

	CASE nState OF

		(*CLEANING CYCLE    --------------------------------------------------------*)
		(*CLEANING CYCLE     --------------------------------------------------------*)
		(*CLEANING CYCLE    --------------------------------------------------------*)

		250:
			iLastState:=nState;

			Block.commands.xStartToCleanOrder:=FALSE;
			Block.commands.xInksOrderCleaning:= TRUE;
			xCloseReliefValve := TRUE; //To force closing the relief valve when ReservoirMode and not cleaning reverseflow
			Block.Status.xCleaningDone:=FALSE;

			ResetKnownPositions;

			nState:= nState+1;

		251:
			iLastState:=nState;
			IF AxisBK.Status.ErrorID=0 THEN
				StopMovements;
				nState:= nState+1;
			END_IF

		252:
			iLastState:=nState;
			IF AllDevicedStopped(ADR(Block), ADR(AxisBK), ADR(IclaBK)) THEN
				IF AxisBK.Status.PowerOn AND AxisBK.Status.PLCopenState.StandStill THEN
					nState:= nState+1;
				END_IF
			END_IF

		253:
			iLastState:=nState;
			//Going Icla To Stop Position
			nState:=nState+1;

		254:
			iLastState:=nState; //the bars go to the drip position.
			// Check Icla Pos because it goes down
			IF Block.In.xIclaSensor THEN
				rMotorAbsPosDesired:= Block.parameters.Motor.rDripBarsPosition;
				MoveAbsolute;
				nState:= nState+1;
			END_IF

		255:
			iLastState:=nState; //the bars go to the drip position.
			// Waiting For Drip Pos Done
			IF ABS(rMotorCurrentPos-rMotorAbsPosDesired)<0.01 THEN
				//Disable cleaning in bar to end ReverseFlow
				Block.commands.xInksOrderCleaning:= FALSE;
				nState:= nState+1;
			END_IF

		256:
			iLastState:=nState;
			//Tray In
			IF NOT Block.In.xTrayIn THEN
				Block.Out.xTrayIn:= TRUE;
			ELSE
				Block.commands.xDripControl:= TRUE;
				nState:= nState+1;
			END_IF

		257:
			iLastState:=nState;
			//Waiting to DripControl End
			IF	NOT Block.commands.xDripControl THEN
				xCloseReliefValve := FALSE;
				nState:= nState+1;
			END_IF

		258:
			iLastState:=nState;
			//Waiting to stabilize Inks
			IF tonStabInksAfterDrip.Q THEN
				nState:= nState + 1;
			END_IF

		259:
			iLastState:=nState;
			//Going To Water Spurt Clean position. Do not protect TrayOut sensor because the bar is over the dripping position
			rMotorAbsPosDesired:= Block.parameters.Motor.rWaterSpurtPosition;
			MoveAbsolute;
			nState:= nState+1;

		260:
			iLastState:=nState;
			//Going To Water Spurt Clean position
			IF ABS(rMotorCurrentPos-rMotorAbsPosDesired)<0.01THEN
				nState:= nState+1;
			END_IF

		261:
			iLastState:=nState;
			//Cleaning motor moving forward
			rIclaAbsPosDesired:= Block.parameters.Icla.rPositionCleanMotorFwd;
			IclaBK.Parameter.MoveAbsolute.Velocity:= Block.parameters.Icla.iCleanMotorSpeedFwd;

			xIclaAbsMovOrder:=TRUE;
			nState:= nState+1;

		262:
			iLastState:=nState;
			//Start water pump activation by position of Icla.
			IF rIclaCurrentPos> Block.parameters.Icla.rFirstHeadPosition THEN
				Block.Out.xCleaningWaterPump:= Block.Status.xIsWaterBlock;
			END_IF

			IF DINT_TO_REAL(IclaBK.Status.iActualPosition) - Block.parameters.Icla.rMinPrintHeadPos > -0.1 THEN
				xIclaAbsMovOrder:= FALSE;
			END_IF

			IF rIclaCurrentPos> Block.parameters.Icla.rLastHeadPosition OR rIclaCurrentPos > Block.parameters.Icla.rPositionCleanMotorFwd - 8.15 THEN
				nState:= nState+1;
			END_IF

		263:
			iLastState:=nState;
			//Stop Water Pump and Change Icla Velocity
			IclaBK.Parameter.MoveAbsolute.Velocity:=500;
			Block.Out.xCleaningWaterPump:= FALSE;

			IF IclaBK.Status.xInPosition THEN
				nState:= nState+1;
			END_IF

		264:
			iLastState:=nState;
			//Wait 3s to depresure water circuit and move Bars to Clean Position
			TON_WaitDepresWater();
			TON_WaitDepresWater.IN:=Block.Status.xIsWaterBlock;
			TON_WaitDepresWater.PT:= T#3s;

			IF NOT Block.Status.xIsWaterBlock OR TON_WaitDepresWater.Q THEN
				TON_WaitDepresWater.IN := FALSE;
				MoveBarsToCleanPosition;
			END_IF

		265:
			CheckAbsolutMovementFinished;

		266:
			iLastState:=nState;
			//Cleaning Motor going to stop position
			xIclaAbsMovOrder:= TRUE;
			rIclaAbsPosDesired:= Block.parameters.Icla.rPositionCleanMotorBwd;
			IclaBK.Parameter.MoveAbsolute.Velocity:=Block.parameters.Icla.iCleanMotorSpeedBwd;

			nState:= nState+1;

		267:
			iLastState:=nState;
			//Start Vacum & Wait Finish Movements
			IF rIclaCurrentPos <= Block.parameters.Icla.rLastHeadPosition THEN
				Block.Out.xVenturi:= Block.parameters.uiCleaningType = 1 OR Block.parameters.uiCleaningType = 2;
			END_IF
			//Stop Venturi
			IF (rIclaCurrentPos <= Block.parameters.Icla.rFirstHeadPosition) THEN
				Block.Out.xVenturi:= FALSE;
			END_IF
			//Remove the xIclaAbsMovOrder to be recepctive for a new positive edge
			IF rIclaCurrentPos <= 70.0  THEN
				xIclaAbsMovOrder:=FALSE;
			END_IF

			//Go to next state to apply the change in Speed
			IF rIclaCurrentPos <= 50.0  THEN
				nState:= nState+1;
			END_IF

		268:
			iLastState:=nState;
			//Change the speed to end the movement
			rIclaAbsPosDesired:= Block.parameters.Icla.rPositionCleanMotorBwd;
			IclaBK.Parameter.MoveAbsolute.Velocity:=500;
			xIclaAbsMovOrder:= TRUE;
			nState:= nState+1;

		269:
			iLastState:=nState;
			//Stop Venturi. If First position is close to 0, stop the venlturi after change speed
			IF (rIclaCurrentPos <= Block.parameters.Icla.rFirstHeadPosition) THEN
				Block.Out.xVenturi:= FALSE;
			END_IF
			//Stopping movement
			IF Block.In.xIclaSensor AND IclaBK.Status.iActualPosition <= 0 THEN
				xIclaAbsMovOrder:= FALSE;
				//Finished cleaning cycle
				Block.Status.xCleaningDone:= TRUE;
				nState:= 0;
			END_IF

	END_CASE

END_ACTION

ACTION MoveAbsolute:
	//Evaluate which speed must be applied
	IF (rMotorCurrentPos>rMotorAbsPosDesired) THEN
		Block.parameters.Motor.rDriveAutoSpeed := Block.parameters.Motor.rAutoSpeedMoveDown;
	ELSE
		//DELOREAN-3070: To set a high speed setpoint for block's motor speed to move up while in printing position
		IF Block.parameters.Motor.xFastSpeedAllowed AND Block.Status.Position.xInPrint THEN
			Block.parameters.Motor.rDriveAutoSpeed := Block.parameters.Motor.rAutoSpeedMoveUpFast;
		ELSE
			Block.parameters.Motor.rDriveAutoSpeed := Block.parameters.Motor.rAutoSpeedMoveUp;
		END_IF
	END_IF
	//Set absolute movement order
	xMotorAbsMovOrder := TRUE;
END_ACTION

ACTION MoveBarsToCleanPosition:
	//Created an action because this code is called from 2 different places
	rMotorAbsPosDesired:= Block.parameters.Motor.rCleanPosition + rOffseCleanMtr;
	MoveAbsolute;
	nState:= nState+1;
END_ACTION

ACTION MoveBarsToCapPosition:
	//Created an action because this code is called from 2 different places
	rMotorAbsPosDesired:= Block.parameters.Motor.rCapPosition;
	MoveAbsolute;
	nState:= nState+1;
END_ACTION

ACTION MoveBarsToCappingPosition:
	//Created an action because this code is called from 2 different places
	rMotorAbsPosDesired:= Block.parameters.Motor.rCappingPosition;
	MoveAbsolute;
	nState:= nState+1;
END_ACTION

ACTION MoveBarsAboveCappingPosition:
	//Created an action because this code is called from 2 different places
	rMotorAbsPosDesired:= Block.parameters.Motor.rCappingPosition + rMoveAboveCapping;
	MoveAbsolute;
	nState:= nState+1;
END_ACTION

ACTION MoveBarsToPrintingPosition:
	//Created an action because this code is called from 2 different places
	rMotorAbsPosDesired:= rCalcPosDesPrint;
	MoveAbsolute;
	nState:= nState+1;
END_ACTION

ACTION CheckAbsolutMovementFinished:
	IF ABS(rMotorCurrentPos-rMotorAbsPosDesired)<0.01 THEN
		nState:= nState+1;
	END_IF
END_ACTION
```

#### ResetCommands.st
```iecst
ACTION ResetBlockCommands:
	Block.commands := stBlockCommandsReseted;
END_ACTION

ACTION ResetHomingBar:

	xMotorHomeOrder := FALSE;
	Block.commands.xBarHomeOrder:=FALSE;
	iTimesStopMovWhileHoming := iTimesStopMovWhileHoming + 1;

	StopBar;

END_ACTION

ACTION ResetHomingIcla:

	//Delete motor orders
	Block.commands.xIclaHomeOrder:=FALSE;
	Block.commands.xIclaHomeOrderInterrupt:=FALSE;
	IclaBK.Command.Home := FALSE;

	StopIcla;

END_ACTION

ACTION ResetCleanCycle:

	Block.commands.Manual.xManIclaBack:=FALSE;
	Block.commands.xDripControl:=FALSE;
	Block.commands.xInksOrderCleaning:= FALSE;
	xCloseReliefValve := FALSE;

	Block.Status.xCleaningDone:=TRUE; //Esto es para que deje de estar en limpieza
	IF BlockPositionPrevious = BLOCKP_CLEANING THEN
		xCleanInterrupt:=TRUE;
	END_IF

	//Stop motors movement and signals
	StopMovements;

END_ACTION

ACTION StopBar:

	AxisBK.Command.Jog.ContinuousNeg:= FALSE;
	AxisBK.Command.Jog.ContinuousPos:= FALSE;
	IF AxisBK.Status.PLCopenState.ContinuousMotion OR AxisBK.Status.PLCopenState.DiscreteMotion THEN
		AxisBK.Command.Move.Halt:=TRUE;
	ELSIF AxisBK.Status.PLCopenState.Homing THEN
		AxisBK.Command.QuickStop:=TRUE;
	ELSIF NOT AxisBK.Status.PLCopenState.Homing THEN
		AxisBK.Command.QuickStop:=FALSE;
	END_IF

END_ACTION

ACTION StopIcla:

	xIclaAbsMovOrder:= FALSE;
	IclaBK.Command.JogFastSpeed:= FALSE;
	IclaBK.Command.JogForward := FALSE;
	IclaBK.Command.JogBackward:= FALSE;
	IF IclaBK.Status.IclaStatus = AXISILE_MOVE_ABSOLUTE OR IclaBK.Status.IclaStatus = AXISILE_JOG THEN
		IclaBK.Command.Stop := TRUE;
	END_IF

END_ACTION

ACTION ResetEdgeCommands:

	IF Block.Status.Position.xGoingToCap OR Block.Status.Position.xInCap THEN
		Block.commands.xToCap := FALSE;
	END_IF
	IF Block.Status.Position.xGoingToPrint OR Block.Status.Position.xInPrint THEN
		Block.commands.xToPrint := FALSE;
	END_IF
	Block.commands.xToCapLab := FALSE;
	Block.commands.xToPrintLab := FALSE;
	Block.commands.xToCleanPosition := FALSE;
	Block.commands.Manual.xToPrintPosition := FALSE;

END_ACTION
```

#### LocalFunctions.fun
```iecst
{REDUND_ERROR} FUNCTION InkBarInBlock : BOOL (*This function returns if the bar determined by the index is in the current block*) (*$GROUP=User,$CAT=User,$GROUPICON=User.png,$CATICON=User.png*)
	VAR_INPUT
		InkIndex : USINT;
		inksArr : REFERENCE TO ARRAY[0..12] OF stInks;
		Block : REFERENCE TO StBlock;
		gIndexBlock : USINT;
	END_VAR
END_FUNCTION

FUNCTION AllDevicedHomed : BOOL
	VAR_INPUT
		Block : REFERENCE TO StBlock;
	END_VAR
END_FUNCTION

FUNCTION AllDevicedStopped : BOOL
	VAR_INPUT
		Block : REFERENCE TO StBlock;
		AxisBK : REFERENCE TO AxisCtrl_typ;
		IclaBK : REFERENCE TO stIcla;
	END_VAR
END_FUNCTION
```

#### InkBarInBlock.st
```iecst
(* This function returns if the bar determined by the index is in the current block *)
FUNCTION InkBarInBlock
	InkBarInBlock := inksArr[InkIndex].parSw.Config.iMappingBar > 0 AND
					(
					(Block.parameters.xLeftHandMachine AND INT_TO_USINT((INT_TO_USINT(inksArr[InkIndex].parSw.Config.iMappingBar)-1) / Block.parameters.Inks.iMaxBlockPrintBars ) = gIndexBlock - 1)	OR
					(Block.parameters.xRightHandMachine AND INT_TO_USINT((INT_TO_USINT(inksArr[InkIndex].parSw.Config.iMappingBar)-1) / Block.parameters.Inks.iMaxBlockPrintBars ) = Block.parameters.iLastBlock - gIndexBlock)
					);

END_FUNCTION
```

#### LogicFunctions.st
```iecst
(* This function returns if the bar determined by the index is in the current block *)
FUNCTION AllDevicedStopped
	AllDevicedStopped := NOT AxisBK.Status.PLCopenState.ContinuousMotion AND
						NOT AxisBK.Status.PLCopenState.Stopping AND
						NOT AxisBK.Status.PLCopenState.DiscreteMotion AND
						IclaBK.Status.iActualVelocity < 5 AND
						NOT Block.Status.Icla.xHoming AND
						NOT Block.Out.xTrayIn AND
						NOT Block.Out.xTrayOut;

END_FUNCTION

(* This function returns TRUE if the cleaning icla motor and the block motor are homed *)
FUNCTION AllDevicedHomed
	AllDevicedHomed := Block.Status.Motor.xBarsHomed AND Block.Status.Icla.xHomed;
END_FUNCTION
```

#### BlockCtrlConst.var
```iecst
VAR CONSTANT
	LIMITPOSINCOHERCLEANMOTOR : REAL := 0.5;
	iHistoryLines : USINT := 20;
END_VAR
```

### Program Logical/ExtPack/BlockCtrl/BlockCtrl_v1/InitBlockCtrl (IEC)

- BlockHomingProcess.graphml - Block States graph (not shown)

- BlockStates.graphml - Block States graph (not shown)

### BlockSim.typ
```iecst
TYPE
	SimBlockCommands_typ : 	STRUCT
		DelayHomingIcla : BOOL; (*With this activated, the SimBlock waits to home the bars until this signal is released*)
		DelayHomingBar : BOOL; (*With this activated, the SimBlock waits to home the bars until this signal is released*)
	END_STRUCT;
	SimBlockParameters_typ : 	STRUCT
		New_Member : BOOL;
	END_STRUCT;
	SimBlock_typ : 	STRUCT
		Commands : SimBlockCommands_typ;
		Parameters : SimBlockParameters_typ;
	END_STRUCT;
END_TYPE
```

### BlockSimIndex.var
```iecst
VAR
	iBlockSimIndex : USINT;
END_VAR
```

### Program Logical/ExtPack/BlockCtrl/BlockSim/BlockSim_v1/InitBlockSim

#### Main.st
```iecst
PROGRAM _CYCLIC

	iBlockSimIndex:= 1;

END_PROGRAM
```

### EFI_General.typ
```iecst
TYPE
	stEFI_AlarmSummary : 	STRUCT
		xAlrSafetySystemGeneral : BOOL;
		xAnyWarning : BOOL;
		xAnyAlarm : BOOL;
		xAlarmCritical : BOOL; (*Out of Auotmatic Mode*)
		xAlarmStop : BOOL;
		xAlarmNonReseteable : BOOL;
		xAlarmReseteable : BOOL;
		xAlarmSound : BOOL;
		iReasonStop : ARRAY[0..1]OF UDINT; (*The reason to move the machine to stop*)
		iReasonWarning : UDINT;
		iReasonCritical : UDINT; (*The reason to move the machine out of auto mode*)
		CurrentReasonStop : ARRAY[0..1]OF UDINT; (*The reason to move the machine to stop*)
		CurrentReasonCritical : UDINT; (*The reason to move the machine out of auto mode*)
		xAlrSafetyCutAir : BOOL; (*Summary alarms to cut the air*)
	END_STRUCT;
	enumEFI_GenMachineState :
		(
		PRINTERGEN_MANUAL,
		PRINTERGEN_ZERO,
		PRINTERGEN_AUTO,
		PRINTERGEN_STARTUP
		);
	enumEFI_MachineState :
		(
		PRINTER_NOT_CLEANING,
		PRINTER_PRINTING,
		PRINTER_CAPPED,
		PRINTER_GOING_TO_CAP,
		PRINTER_GOING_TO_PRINT,
		PRINTER_CLEANING
		);
	enumEFI_MachineAutoStatesMode :
		(
		AUTO_NOT_VALID,
		AUTO_PRODUCTION,
		AUTO_BYPASS,
		AUTO_STOP,
		AUTO_LABORATORY,
		AUTO_JAMRECOVERY
		);
	enumEFI_SafetySignals :
		(
		SAFETY_ESTOP_CONNECTED,
		SAFETY_ESTOP_CALCULATED
		);
	stEFI_MachineAutoModes : 	STRUCT
		xLaboratory : BOOL; (*Laboratory Mode*)
		xStop : BOOL; (*Stop Mode*)
		xProduction : BOOL; (*Production/AutoRun Mode*)
		xBypass : BOOL; (*Bypass Mode*)
		xPause : BOOL; (*Pause Mode*)
		xJamRecovery : BOOL; (*JamRecovery Mode*)
		xProdORByPass : BOOL; (*Combined BOOL to better reading. Production OR ByPass Mode*)
		xProdORLab : BOOL; (*Combined BOOL to better reading. Production OR Laboratory Mode*)
	END_STRUCT;
	MotorDirection_enum :
		(
		MOTOR_POSITIVE := 0, (*This is the value expected in AxisCtrl. 0 for Postive*)
		MOTOR_NEGATIVE := 1 (*This is the value expected in AxisCtrl. 1 for Negative*)
		);
	LineStatus_enum :
		(
		LINE_NOT_POWERED, (*This is the starting state when starting to allow StatusChange to be receptive*)
		LINE_ERROR,
		LINE_PREPARING_EMPTYBELT,
		LINE_PREPARING_PRINT,
		LINE_PREPARING_CLEANPH,
		LINE_PREPARING_CLEANBELT,
		LINE_STARTING_PRINTING,
		LINE_STARTING_CLEANINGPH,
		LINE_STARTING_CLEANINGBELT,
		LINE_BELT_EMPTYING,
		LINE_CLEANED,
		LINE_STARTING_EMPTYBELT,
		LINE_IDLE,
		LINE_PRINTING,
		LINE_PAUSING,
		LINE_PAUSED,
		LINE_CLEANINGPH,
		LINE_CLEANINGBELT,
		LINE_CONTROLLED_STOP,
		LINE_STOPPED,
		LINE_NOT_INITIALIZED,
		LINE_INITIALIZING,
		LINE_POWERING_OFF
		);
	EFI_version_typ : 	STRUCT
		iVersion0 : INT;
		iVersion1 : INT;
		iVersion2 : INT;
		iVersion3 : INT;
	END_STRUCT;
	CommsNetworkType_enum :
		(
		COMMS_UNDEFINED,
		COMMS_POWERLINK,
		COMMS_CANOPEN
		);
	CanOpenResetCommsState_enum :
		(
		COCOMSR_UNDEFINED,
		COCOMSR_COMMUNICATING,
		COCOMSR_COMMSERROR,
		COCOMSR_RESETTING,
		COCOMSR_WAITINGTOBERESETTED,
		COCOMSR_RESETTING_ERROR
		);
	StGeneral_States_Mode : 	STRUCT
		xManual : {REDUND_UNREPLICABLE} BOOL; (*State to define Manual Mode*)
		xZero : BOOL; (*State to define Zero Mode*)
		xAuto : BOOL; (*State to define Auto Mode*)
		xStartUp : BOOL; (*State to define StartUp Mode*)
	END_STRUCT;
	LineControlStatusSummarized : 	STRUCT
		xLineEmpty : BOOL;
		xIdle : BOOL;
		xStopped : BOOL;
		xControlStopping : BOOL;
		xErrorStopping : BOOL;
		xCleaning : BOOL;
		xEmptyingBelts : BOOL;
		xPausing : BOOL;
		xCleaningBelt : BOOL;
		xPrinting : BOOL;
	END_STRUCT;
	InvType_enum :
		(
		INV_BR,
		INV_ABB
		);
	OpcUaCommsState :
		(
		OPCUA_IDLE,
		OPCUA_CONNECTING,
		OPCUA_GETTING_NAMESPACE,
		OPCUA_GETTING_HANDLE,
		OPCUA_EXECUTING,
		OPCUA_PAUSED,
		OPCUA_RELEASINSG_HANDLE,
		OPCUA_DISCONNECTING,
		OPCUA_FAULTED
		);
	SimDryerType :
		(
		SIM_DRYER_NOZ2_NIR_ARCLAMP := 1,
		SIM_DRYER_NOZ2_NIR := 2
		);
	ChillerStatus_enum :
		(
		CHILLER_OFF,
		CHILLER_STARTING,
		CHILLER_RUNNING,
		CHILLER_STOPPING,
		CHILLER_FAULT
		);
END_TYPE
```

### Program Logical/ExtPack/EFILib/EFILib_v1/ConvertFun

#### Constants.var
```iecst
VAR CONSTANT
	NAN_VALUE_UDINT : UDINT := 16#FFC00000; (*16#FFC00000 is the bit pattern of the NaN value for a REAL variable. It must be copied to a REAL variable using the memcpy FB*)
END_VAR
```

#### SECONDS_TO_MILLIS.st
```iecst
(* TODO: Add your comment here *)
FUNCTION SECONDS_TO_MILLIS
	SECONDS_TO_MILLIS := iSeconds*1000;
END_FUNCTION
```

#### SECONDS_TO_TIME.st
```iecst
(* TODO: Add your comment here *)
FUNCTION SECONDS_TO_TIME

	SECONDS_TO_TIME := UDINT_TO_TIME(SECONDS_TO_MILLIS(iSeconds));	//Time conversion needs

END_FUNCTION
```

#### TIME_TO.st
```iecst
(* TODO: Add your comment here *)
FUNCTION TIME_TO_MINUTES

	TIME_TO_MINUTES := REAL_TO_INT(TIME_TO_REAL(tiTimeValue)/1000/60); //Value in time are ms, and here we convert it to minutes

END_FUNCTION

(* TODO: Add your comment here *)
FUNCTION TIME_TO_SECONDS

	TIME_TO_SECONDS := TIME_TO_UDINT(tiTimeValue)/1000; //Value in time are ms, and here we convert it to seconds

END_FUNCTION

(* TODO: Add your comment here *)
FUNCTION TIME_TO_SECONDS_COMS

	TIME_TO_SECONDS_COMS := UDINT_TO_UINT(TIME_TO_UDINT(tiTimeValue)/1000); //Value in time are ms, and here we convert it to seconds

END_FUNCTION

(* TODO: Add your comment here *)
FUNCTION TIME_TO_MILLISECONDS

	TIME_TO_MILLISECONDS := TIME_TO_UDINT(tiTimeValue); //Value in time are ms, and here we convert it directly to milliseconds in UDINT

END_FUNCTION

(* TODO: Add your comment here *)
FUNCTION TIME_TO_MILLISECONDS_COMS

	TIME_TO_MILLISECONDS_COMS := TIME_TO_UINT(tiTimeValue); //Value in time are ms, and here we convert it directly to milliseconds in UINT

END_FUNCTION
```

### Library Logical/ExtPack/EFILib/EFILib_v1/FBs

#### EFILib.typ
```iecst
(*********************************************************************
* Drive Unit Manager
*********************************************************************)

TYPE
	MD_CalculationType :
		(
		CALC_HOMEPOS_PULSES,
		CALC_HOMEPOS_MM, (*Position in mm*)
		CALC_JOGSPEED_PULSES,
		CALC_JOGSPEED_MM, (*JogSpeed in mm/s*)
		CALC_SPEED_MMIN_PULSES,
		CALC_SPEED_MMIN, (*Speed in m/min*)
		CALC_SPEED_PULSES,
		CALC_SPEED_MM, (*Speed in mm/s*)
		CALC_SPEED_REVMIN_MMIN,
		CALC_POS_PULSES,
		CALC_POS_MM, (*Position in mm*)
		CALC_ACC_PULSES,
		CALC_ACC_MM, (*Acceleration in mm/s^2*)
		CALC_DEC_PULSES,
		CALC_DEC_MM (*Deceleration in mm/s^2*)
		);
	MD_TransmissionType :
		(
		TRANS_UNDEFINED,
		TRANS_SCREW_PITCH,
		TRANS_LINEAL_DIAMETER,
		TRANS_LINEAL_PERIMETER
		);
	MC_TransLinealDiameter_typ : 	STRUCT
		PulsesPerTurn : UDINT; (*Units considered by the drive for 1 turn*)
		GearBox : REAL; (*Reduction :1*)
		Diameter : REAL; (*Diameter in mm*)
	END_STRUCT;
	MC_TransLinealPerimeter_typ : 	STRUCT
		PulsesPerTurn : UDINT; (*Units considered by the drive for 1 turn*)
		GearBox : REAL; (*Reduction :1*)
		Perimeter : REAL; (*Perimeter in mm*)
	END_STRUCT;
	MC_TransScrewPitch_typ : 	STRUCT
		PulsesPerTurn : UDINT; (*Units considered by the drive for 1 turn*)
		GearBox : REAL; (*Reduction :1*)
		Pitch : REAL; (*Pitch in mm*)
	END_STRUCT;
	MC_DriveUnitManager : 	STRUCT
		TransmissionType : MD_TransmissionType := TRANS_UNDEFINED; (*Used to avoid problems if DriveUnit is executed but not configured*)
		LinealDiameter : MC_TransLinealDiameter_typ;
		LinealPerimeter : MC_TransLinealPerimeter_typ;
		ScrewPitch : MC_TransScrewPitch_typ;
	END_STRUCT;
	AnalogProcessSimType_enum :
		(
		ANALOGSIM_LINEAR_POS, (*If no action, the signal raises*)
		ANALOGSIM_LINEAR_NEG, (*If no action, the signal goes down*)
		ANALOGSIM_EXPONENTIAL_POS, (*If no action, the signal raises*)
		ANALOGSIM_EXPONENTIAL_NEG (*If no action, the signal goes down*)
		);
END_TYPE
```

#### Global_Constant.var
```iecst
VAR CONSTANT
	GC_CONFIG_1BK2BAR : STRING[80] := '1BK2Bar'; (*Config for Shield*)
	GC_CONFIG_1BK2BAR_ID : USINT := 12; (*Config for Shield*)
	GC_CONFIG_1BK8BAR_NOZ2 : STRING[80] := '1BK8Bar_Noz2'; (*Config for 1 block and 8 bars Nozomi2*)
	GC_CONFIG_1BK8BAR_NOZ2_ID : USINT := 30; (*Config for Nozomi2*)
	GC_CONFIG_1BK8BAR_NOZ2_AQ : STRING[80] := '1BK8Bar_Noz2_AQ'; (*Config for 1 block and 8 bars Nozomi2 Water*)
	GC_CONFIG_1BK8BAR_NOZ2_AQ_ID : USINT := 70; (*Config for Nozomi2 Water*)
	GC_CONFIG_PLCDIAGNOSIS : STRING[80] := 'PlcDiagnosis'; (*Config for PlcDiagnosis *)
	GC_CONFIG_PLCDIAGNOSIS_ID : USINT := 100; (*Config for PlcDiagnosis *)
	GC_CONFIG_1BK10BAR_MECANO : STRING[80] := '1BK10Bar_Mecano'; (*Config for 1 block and 10 bars Mecano*)
	GC_CONFIG_1BK10BAR_MECANO_ID : USINT := 40; (*Config for Mecano*)
	GC_CONFIG_1BK7BAR_CUBE : STRING[80] := '1BK7Bar_Cube'; (*Config for 1 block and 7 bars Cube*)
	GC_CONFIG_1BK7BAR_CUBE_ID : USINT := 61; (*Config for Cube*)
	GC_CONFIG_2BK12BAR : STRING[80] := '2BK12Bar'; (*Config for P4*)
	GC_CONFIG_2BK12BAR_ID : USINT := 11; (*Config for P4*)
	GC_CONFIG_BM_1BK8BAR : STRING[80] := 'BM_1BK8Bar'; (*Config for 1 block and 8 bars building materials machines*)
	GC_CONFIG_BM_1BK8BAR_ID : USINT := 13; (*Config for S1400 or P5*)
	GC_CONFIG_DRYER_NOZ2 : STRING[80] := 'Dryer'; (*Config for Dryer*)
	GC_CONFIG_DRYER_NOZ2_ID : USINT := 53; (*Config for Dryer Nozomi2*)
	GC_CONFIG_SIMDRYER_NOZ2 : STRING[80] := 'SimDryer'; (*Config for Dryer Simulation*)
	GC_CONFIG_SIMDRYER_NOZ2_ID : USINT := 54; (*Config for Dryer Nozomi2 Simulation*)
	GC_CONFIG_SIMTEST : STRING[80] := 'SimTests'; (*Config for Simulation*)
	GC_CONFIG_SIMTEST_ID : USINT := 10; (*Config for Simulation*)
	GC_CONFIG_INKBOX : STRING[80] := 'InkBox'; (*Config for InkBox*)
	GC_CONFIG_INKBOX_ID : USINT := 91; (*Config for InkBox*)
	GC_CONFIG_INKBOX_SIM_ID : USINT := 92; (*Config for InkBox in SIMULATION*)
	gc_diNumMaxManiobrasPDoblada : DINT := 150;
	GC_DTP_BYPASS : INT := 1; (*DTP Line Mode = 1*)
	GC_DTP_RUN : INT := 0; (*DTP Line Mode = 0*)
	GC_DTP_STOP : INT := 2; (*DTP Line Mode = 2*)
	GC_FIRST_BLOCK : USINT := 1;
	GC_MIN_OFFSET_BLOCK : REAL := 0.0;
	GC_MIN_PIECES_TO_CLEAN : INT := 10; (*// Número mínimo de piezas hasta realizar la limpieza de la barra por piezas*)
	gc_rMinSpeedToStart : REAL := 1.0; (*Minimum speed to consider movement in the position arrays*)
	GC_TEMP_SP_PRINTHEADS : REAL := 22.0; (*Set Point temperature for printheads*)
	gc_tiTesperaAlarmaAire : TIME := T#1S;
	gc_tiTpoAlrManiobrasPDoblada : TIME := T#900S;
	GC_UNITS_BY_REV_DRIVE : UDINT := 1000; (*Vertical Motor Units By Revolution*)
	MAX_EXTERNAL_DEVICES : USINT := 20; (*To define the array*)
	MAX_LAST_BLOCK : USINT := 2; (*Do not use in program. Just here to define the array*)
	MAX_LAST_SIMPLEBLOCK : USINT := 1; (*Do not use in program. Just here to define the array*)
	MAX_LAST_INK : USINT := 12; (*To define the array*)
	MAX_LAST_JAMDEVICE : USINT := 16; (*To define the array*)
	MAX_LAST_JAMSENSOR : USINT := 4; (*To define the array*)
	MAX_LAST_MOTOR_BLOWER : USINT := 2;
	MAX_LAST_NON_CRASH : USINT := 2;
	MAX_LAST_CURING_LED : USINT := 3;
	MAX_LAST_NIR_MODULES : USINT := 2;
	MAX_EHD_ADJUST_SYSTEMS : USINT := 2; (*Maximum number of adjustments systems used in by the edge hold down*)
	MAX_EHD_MOTORS_PER_ADJUST_SYS : USINT := 2; (*Maximum number of motors used in an Edge hold down's adjustment system*)
	MAX_LAST_ICLA_MOTOR : USINT := 8; (*To define the array*)
	MAX_LAST_NSENSOR : USINT := 8; (*To define the array*)
	MAX_LAST_TRANS_VACUUM : USINT := 5; (*To define the array*)
	MAX_LAST_INVERTER : USINT := 6; (*To define the array*)
	MAX_LAST_GEW_ARCLAMPS : USINT := 2; (*To define the array*)
	MAX_LAST_INK_CABINET : USINT := 4; (*To define the array*)
	MAX_LAST_INK_IN_CABINET : USINT := 2; (*To define the array*)
	MAX_LAST_CURING_LED_LAMP : USINT := 16;
	MAX_LAST_CHECKMEDIA : USINT := 2;
	MAX_LAST_CHILLER : USINT := 2;
	MAX_LAST_SIGNAL : USINT := 16; (*Quantity of signals in the mapping structure arrays*)
	MIN_CLEANING_BY_TIME : TIME := T#5m; (*//   Minimo tiempo hasta realizar la limpieza de la barra  (en minutos)*)
	MIN_CLEANING_STOPPED : TIME := T#5m; (*//   Minimo tiempo hasta realizar la limpieza de la barra  (en minutos)*)
	MAX_LAST_REQUIRED_FUNCTION_CARD : USINT := 3;
	MAX_LAST_ADJUSTMENT_SYSTEM : USINT := 2;
	MAX_LAST_HEATER_PSU_AC_OK : USINT := 3;
	MAX_LAST_HEATER_PSU_DC_OK : USINT := 3;
	MAX_LAST_PH_PSU : USINT := 6;
END_VAR
```

#### ThicknessCtrlPublicConst.var
```iecst
VAR CONSTANT
	TOTAL_THICKNESS_SECTIONS : USINT := 5;
	iMAXTRACKINGARRAY : UINT := 3000;
	iMAXHEIGHTARRAY : UINT := 800;
	iMAXMEDIAPRESENTARRAY : UINT := 500;
END_VAR
```

#### FBs.fun
```iecst
FUNCTION_BLOCK AutoResetSound
	VAR_INPUT
		xAlarm : BOOL;
		xSilence : BOOL;
	END_VAR
	VAR_OUTPUT
		xAlarmSound : BOOL;
	END_VAR
	VAR
		fbRiseUpAlarm : R_TRIG;
	END_VAR
END_FUNCTION_BLOCK

FUNCTION_BLOCK FbCleanDelayControl
	VAR_INPUT
		T_delay_L1 : TIME; (*	// Line 1 TIME delay  *)
		T_delay_L2 : TIME; (*	// Line 2 TIME delay *)
		Start : BOOL; (*//Sequence start*)
		Doble : BOOL; (*//Doble line*)
		t_Gap : TIME; (*//Gap TIME*)
	END_VAR
	VAR_OUTPUT
		End : BOOL; (*//Delay end*)
		Out_L1 : BOOL; (*//Stop output line 1*)
		Out_L2 : BOOL; (*	//Stop output line 2*)
	END_VAR
	VAR
		T_delay1 : TIME;
		T_delay2 : TIME;
		TON_1 : TON;
		TON_5 : TON;
		TON_4 : TON;
		TON_6 : TON;
		TON_12 : TON;
		TON_14 : TON;
		TON_13 : TON;
		TON_15 : TON;
		TON_9 : TON;
		TON_16 : TON;
		TON_0 : TON;
		TON_3 : TON;
		TON_2 : TON;
	END_VAR
END_FUNCTION_BLOCK

FUNCTION_BLOCK MotorSpeedCalculation (*Motor Speed calculation*)
	VAR_INPUT
		xEnable : BOOL;
		iSpSpeed : INT; (*Speed in meter per minute*)
		uiReductor : UINT := 1; (*Reductor ratio*)
		uiRolllerPerimeter : UINT := 10; (*Perimeter belt roller, Length roller in mm*)
		xPrinterDirection : BOOL; (* 0=Right,1= Left*)
		rUnitsAtTheLoad : REAL; (*1 rev motor are 1000 Units at the load*)
	END_VAR
	VAR_OUTPUT
		xChange : BOOL;
		rSpeedMotor : REAL; (*Output speed in mXmin*)
	END_VAR
	VAR
		Aux : REAL;
		m_rpm : REAL := 1;
	END_VAR
END_FUNCTION_BLOCK

FUNCTION_BLOCK SetCalcVelocity (*TODO: Add your comment here*) (*$GROUP=User,$CAT=User,$GROUPICON=User.png,$CATICON=User.png*)
	VAR_INPUT
		xEnMov : BOOL;
		rSpeed : REAL; (*Speed in m/min*)
		rReduction : REAL := 0.0; (*GearBox ratio*)
		rAxisDiamter : REAL := 0.0; (*Length of a turn in mm*)
		rUnitsAtTheLoad : REAL; (*Units configured in the drive for 1 turn*)
	END_VAR
	VAR_OUTPUT
		xChange : BOOL; (*Signal of change in the speed setpint*)
		rSpeedInUnits : REAL;
	END_VAR
	VAR
		rLastSpeedInUnits : REAL := 0; (*Initilialize is important!!!!!!!!!!!!!!!*)
		zzEdge00000 : BOOL;
	END_VAR
END_FUNCTION_BLOCK

FUNCTION_BLOCK GetCalcVelocity (*TODO: Add your comment here*) (*$GROUP=User,$CAT=User,$GROUPICON=User.png,$CATICON=User.png*)
	VAR_INPUT
		xEn : BOOL; (*	// Enable lectura*)
		xValid : BOOL; (*	// Recepción de la velocidad del motor ok*)
		diVelocidad_RPM : DINT; (*// Valor leido en RPM*)
		uiReductor : UINT; (*// Relacion del reductor con tres decimales*)
		uiEje : UINT; (*	// Recorrido de una vuelta de eje en mm*)
	END_VAR
	VAR_OUTPUT
		iVel_lin : DINT; (*// Velocidad en metros/min*)
	END_VAR
	VAR
		rValor : REAL;
		rm_rpm : REAL;
	END_VAR
END_FUNCTION_BLOCK

FUNCTION_BLOCK Blink
	VAR_INPUT
		T_Blink : TIME;
	END_VAR
	VAR_OUTPUT
		Out : BOOL;
	END_VAR
	VAR
		T_OFF : TON;
		T_ON : TON;
		VAR1 : BOOL;
	END_VAR
END_FUNCTION_BLOCK

FUNCTION_BLOCK ComandBoolT (*TODO: Add your comment here*) (*$GROUP=User,$CAT=User,$GROUPICON=User.png,$CATICON=User.png*)
	VAR_IN_OUT
		In : BOOL; (*//Valor de entrada*)
		Com : INT; (*//Para poner el comando a -1*)
	END_VAR
	VAR
		Contador : INT;
	END_VAR
END_FUNCTION_BLOCK

FUNCTION_BLOCK BlinkOnOff (*TODO: Add your comment here*) (*$GROUP=User,$CAT=User,$GROUPICON=User.png,$CATICON=User.png*)
	VAR_INPUT
		xEnable : BOOL;
		tTimeOn : TIME;
		tTimeOff : TIME;
	END_VAR
	VAR_OUTPUT
		xOutput : BOOL;
	END_VAR
	VAR
		TON_1 : TON;
		TON_2 : TON;
	END_VAR
END_FUNCTION_BLOCK
(*Pending TO implememnt
FUNCTION_BLOCK InterfaceNetworkCommands It sends commands by CanOpen Interface to reset node
	VAR_INPUT
		xEnable : BOOL := FALSE; Enable action in this FB
		xModuleOk : BOOL := TRUE; It sets state of the module to check
		arrayInterfaceNetwork : STRING[3] := 'IF7'; This var contains the interface network type. Interface Network types forType of network:RS232 interface (IF1), Ethernet interface (IF2), POWERLINK interface (IF3), USB interfaces (IF4 and IF5) and CAN bus interface (IF7)
		iIdNode : UINT := 180; Node Identifier
		command : UINT := 3; commnad coRESET_NODE by default is reset node as enum defined in AsCanOpen
	END_VAR
	VAR_OUTPUT
		statusNode : BOOL := TRUE; ERROR or OK state
	END_VAR
END_FUNCTION_BLOCK*)
(*Function to simulate an analog process and be able to run programs in Simulation
PVnext := PVprevious - A + B * ActionControl*)

FUNCTION_BLOCK SimAnalogProcess
	VAR_INPUT
		AnalogType : AnalogProcessSimType_enum := ANALOGSIM_LINEAR_NEG;
		rA : REAL; (*Behavior Constant. Fixed desdent of PV without control action*)
		rB : REAL; (*Behavior Constant. Increment of PV with control action*)
		rMaxValue : REAL;
		rMinValue : REAL;
		rInitialValue : REAL;
		rActionControl : REAL;
		rNewPresentValue : REAL;
		xUseNewValue : BOOL := FALSE;
	END_VAR
	VAR_OUTPUT
		rPresentValue : REAL;
	END_VAR
	VAR
		xStarted : BOOL := FALSE;
		rSignalPerct : REAL; (*Current signal percentaje in the limits*)
		zzEdge00000 : BOOL;
	END_VAR
END_FUNCTION_BLOCK

{REDUND_ERROR} FUNCTION_BLOCK DriveUnitMngr (*Funtion Block to Manage Drive Units from and to the Drive*) (*$GROUP=User,$CAT=User,$GROUPICON=User.png,$CATICON=User.png*)
	VAR_INPUT
		Calculation : MD_CalculationType;
		JogSpeedDesired : {REDUND_UNREPLICABLE} REAL; (*Value in mm/s of the desired position*)
		SpeedMminDesired : {REDUND_UNREPLICABLE} REAL; (*Value in m/min of the desired Speed*)
		SpeedDesired : {REDUND_UNREPLICABLE} REAL; (*Value in mm/s of the desired Speed*)
		AccelerationDesired : {REDUND_UNREPLICABLE} REAL; (*Value in mm/s^2 of the desired Acceleration*)
		DecelerationDesired : {REDUND_UNREPLICABLE} REAL; (*Value in mm/s^2 of the desired Acceleration*)
		HomePositionDesired : {REDUND_UNREPLICABLE} REAL; (*Value in mm of the desired position*)
		PositionDesired : {REDUND_UNREPLICABLE} REAL; (*Value in mm of the desired position*)
		PulsesAccelerationDevice : {REDUND_UNREPLICABLE} REAL; (*Acceleration in pulses/s2*)
		PulsesDecelerationDevice : {REDUND_UNREPLICABLE} REAL; (*Deceleration in pulses/s2*)
		PulsesSpeedDevice : {REDUND_UNREPLICABLE} REAL; (*Current speed in pulses/s*)
		RevMinSpeedDevice : {REDUND_UNREPLICABLE} REAL; (*Current speed in rev/min*)
		pulsesDevice : {REDUND_UNREPLICABLE} REAL; (*Current position in pulses *)
		TransmissionData : MC_DriveUnitManager; (*Transmission data*)
	END_VAR
	VAR_OUTPUT
		pulsesJogSpeedDesired : REAL; (*Value in pulses/s of the desired speed*)
		pulsesSpeedDesired : REAL; (*Value in pulses/s of the desired speed*)
		pulsesAccelerationDesired : REAL; (*Value in pulses/s^2 of the desired acceleration*)
		pulsesDecelerationDesired : REAL; (*Value in pulses/s^2 of the desired acceleration*)
		pulsesHomePositionDesired : REAL; (*Value in pulses of the desired position*)
		pulsesPositionDesired : REAL; (*Value in pulses of the desired position*)
		mmAcceleration : REAL; (*Value in mm/s^2 of the desired acceleration*)
		mmDeceleration : REAL; (*Value in mm/s^2 of the desired acceleration*)
		SpeedDevice : REAL; (*Current Speed in mm/s*)
		SpeedRpmToMmin : REAL; (*Current Speed in m/min*)
		SpeedMminDevice : REAL; (*Current Speed in m/min*)
		PositionDevice : REAL; (*Current position in mm*)
		mmToPulses : REAL := 1.0;
		mmToTurn : REAL := 1.0;
	END_VAR
	VAR
		JogSpeedDesiredCopy : REAL := -1; (*Value in mm of the desired speed. Initialized to a value not allowed to force a first execution*)
		SpeedMminDesiredCopy : REAL := -1; (*Value in m/min of the desired speed. Initialized to a value not allowed to force a first execution*)
		SpeedDesiredCopy : REAL := -1; (*Value in mm/2 of the desired speed. Initialized to a value not allowed to force a first execution*)
		AccelerationDesiredCopy : REAL := -1; (*Value in mm/s^2 of the desired acceleration. Initialized to a value not allowed to force a first execution*)
		DecelerationDesiredCopy : REAL := -1; (*Value in mm/s^2 of the desired acceleration. Initialized to a value not allowed to force a first execution*)
		HomePositionDesiredCopy : REAL := -1; (*Value in mm of the desired position. Initialized to a value not allowed to force a first execution*)
		PositionDesiredCopy : REAL := -1; (*Value in mm of the desired position. Initialized to a value not allowed to force a first execution*)
		pulsesAccelerationDeviceCopy : REAL := -1; (*Acceleration in pulses*)
		pulsesDecelerationDeviceCopy : REAL := -1; (*Deceleration in pulses*)
		pulsesSpeedDeviceCopy : REAL := -1; (*Current speed in pulses/s. Initialized to a value not allowed to force a first execution*)
		RevMinSpeedDeviceCopy : REAL := -1; (*Current speed in rev/min*)
		pulsesDeviceCopy : REAL := -1; (*Current position in pulses. Initialized to a value not allowed to force a first execution*)
		mmToPulsesCopy : REAL := -1; (*Initialized to a value not allowed to force a first execution*)
		TransDataCopy : MC_DriveUnitManager;
	END_VAR
END_FUNCTION_BLOCK
```

#### AutoResetSound.st
```iecst
(* TODO: Add your comment here *)
FUNCTION_BLOCK AutoResetSound

	fbRiseUpAlarm(CLK:=xAlarm);
	IF fbRiseUpAlarm.Q THEN xAlarmSound:=TRUE; END_IF
	IF xSilence OR NOT xAlarm THEN xAlarmSound:=FALSE; END_IF

END_FUNCTION_BLOCK
```

#### DriveUnitMngr.st
```iecst
(* Funtion Block to Manage Drive Units from and to the Drive *)
FUNCTION_BLOCK DriveUnitMngr

(*	PositionDesired	REAL	VAR_INPUT
	pulsesDevice	DINT	VAR_INPUT
	TransmissionData	MC_DriveUnitManager	VAR_INPUT
	pulsesPositionDesired	DINT		VAR_OUTPUT
	PositionDevice	REAL		VAR_OUTPUT
	TransDataCopy	MC_DriveUnitManager
	mmToPulses	REA	VAR

*)

	//RETURN if the FB is not configured
	IF TransmissionData.TransmissionType = TRANS_UNDEFINED THEN
		RETURN;
	END_IF

	CASE TransmissionData.TransmissionType OF

		TRANS_SCREW_PITCH:
			IF 	TransDataCopy.ScrewPitch.GearBox <> TransmissionData.ScrewPitch.GearBox OR
				TransDataCopy.ScrewPitch.Pitch <> TransmissionData.ScrewPitch.Pitch OR
				TransDataCopy.ScrewPitch.PulsesPerTurn <> TransmissionData.ScrewPitch.PulsesPerTurn
																					THEN
					TransmissionData.ScrewPitch.PulsesPerTurn := MAX(TransmissionData.ScrewPitch.PulsesPerTurn, 2);
					TransmissionData.ScrewPitch.Pitch := MAX(TransmissionData.ScrewPitch.Pitch, 2);
					IF TransmissionData.ScrewPitch.GearBox=0 THEN TransmissionData.ScrewPitch.GearBox:=1; END_IF

					mmToTurn := TransmissionData.ScrewPitch.GearBox/TransmissionData.ScrewPitch.Pitch;
					mmToPulses:=UDINT_TO_REAL(TransmissionData.ScrewPitch.PulsesPerTurn)*mmToTurn;

					//Initialize the value of the copys to be sure to recalculate after a parameters update
					pulsesDeviceCopy:=1.0E-10;
					PositionDesiredCopy:=1.0E-10;
					HomePositionDesiredCopy:=1.0E-10;
					JogSpeedDesiredCopy:=1.0E-10;
					SpeedDesiredCopy:=1.0E-10;
					AccelerationDesiredCopy:=1.0E-10;
					DecelerationDesiredCopy:=1.0E-10;
					pulsesSpeedDeviceCopy:=1.0E-10;
					RevMinSpeedDeviceCopy:=1.0E-10;
					pulsesAccelerationDeviceCopy:=1.0E-10;
					pulsesDecelerationDeviceCopy:=1.0E-10;

			END_IF

		TRANS_LINEAL_DIAMETER:
			IF 	TransDataCopy.LinealDiameter.GearBox <> TransmissionData.LinealDiameter.GearBox OR
				TransDataCopy.LinealDiameter.Diameter <> TransmissionData.LinealDiameter.Diameter OR
				TransDataCopy.LinealDiameter.PulsesPerTurn <> TransmissionData.LinealDiameter.PulsesPerTurn
																					THEN
					TransmissionData.LinealDiameter.PulsesPerTurn:= MAX(TransmissionData.LinealDiameter.PulsesPerTurn, 2);
					TransmissionData.LinealDiameter.Diameter:= MAX(TransmissionData.LinealDiameter.Diameter, 2);
					IF TransmissionData.LinealDiameter.GearBox=0 THEN TransmissionData.LinealDiameter.GearBox:=1; END_IF

					mmToTurn := TransmissionData.LinealDiameter.GearBox/(brmPI*TransmissionData.LinealDiameter.Diameter);
					mmToPulses:=UDINT_TO_REAL(TransmissionData.LinealDiameter.PulsesPerTurn)*mmToTurn;

					//Initialize the value of the copys to be sure to recalculate after a parameters update
					pulsesDeviceCopy:=1.0E-10;
					PositionDesiredCopy:=1.0E-10;
					HomePositionDesiredCopy:=1.0E-10;
					JogSpeedDesiredCopy:=1.0E-10;
					SpeedDesiredCopy:=1.0E-10;
					AccelerationDesiredCopy:=1.0E-10;
					DecelerationDesiredCopy:=1.0E-10;
					pulsesSpeedDeviceCopy:=1.0E-10;
					RevMinSpeedDeviceCopy:=1.0E-10;
					pulsesAccelerationDeviceCopy:=1.0E-10;
					pulsesDecelerationDeviceCopy:=1.0E-10;

			END_IF

		TRANS_LINEAL_PERIMETER:
			IF 	TransDataCopy.LinealPerimeter.GearBox <> TransmissionData.LinealPerimeter.GearBox OR
				TransDataCopy.LinealPerimeter.Perimeter <> TransmissionData.LinealPerimeter.Perimeter OR
				TransDataCopy.LinealPerimeter.PulsesPerTurn <> TransmissionData.LinealPerimeter.PulsesPerTurn
																					THEN
					TransmissionData.LinealPerimeter.PulsesPerTurn:= MAX(TransmissionData.LinealPerimeter.PulsesPerTurn, 2);
					TransmissionData.LinealPerimeter.Perimeter:= MAX(TransmissionData.LinealPerimeter.Perimeter, 2);
					IF TransmissionData.LinealPerimeter.GearBox=0 THEN TransmissionData.LinealPerimeter.GearBox:=1; END_IF

					mmToTurn := TransmissionData.LinealPerimeter.GearBox/TransmissionData.LinealPerimeter.Perimeter;
					mmToPulses:=UDINT_TO_REAL(TransmissionData.LinealPerimeter.PulsesPerTurn)*mmToTurn;

					//Initialize the value of the copys to be sure to recalculate after a parameters update
					pulsesDeviceCopy:=1.0E-10;
					PositionDesiredCopy:=1.0E-10;
					HomePositionDesiredCopy:=1.0E-10;
					JogSpeedDesiredCopy:=1.0E-10;
					SpeedDesiredCopy:=1.0E-10;
					AccelerationDesiredCopy:=1.0E-10;
					DecelerationDesiredCopy:=1.0E-10;
					pulsesSpeedDeviceCopy:=1.0E-10;
					RevMinSpeedDeviceCopy:=1.0E-10;
					pulsesAccelerationDeviceCopy:=1.0E-10;
					pulsesDecelerationDeviceCopy:=1.0E-10;

			END_IF

	END_CASE;

	//To avoid NotaNumber messages
	IF mmToPulses=0 THEN
		RETURN;
	END_IF

	CASE Calculation OF
		CALC_POS_MM:
			IF pulsesDevice<>pulsesDeviceCopy OR mmToPulsesCopy<>mmToPulses THEN
				PositionDevice:=pulsesDevice/mmToPulses;
				pulsesDeviceCopy:=pulsesDevice;
			END_IF;

		CALC_POS_PULSES:
			IF PositionDesired<>PositionDesiredCopy OR mmToPulsesCopy<>mmToPulses THEN
				pulsesPositionDesired:=PositionDesired*mmToPulses;
				PositionDesiredCopy:=PositionDesired;
			END_IF;

		CALC_HOMEPOS_PULSES:
			IF HomePositionDesired<>HomePositionDesiredCopy OR mmToPulsesCopy<>mmToPulses THEN
				pulsesHomePositionDesired:=HomePositionDesired*mmToPulses;
				HomePositionDesiredCopy:=HomePositionDesired;
			END_IF;

		CALC_JOGSPEED_PULSES:
			IF JogSpeedDesired<>JogSpeedDesiredCopy OR mmToPulsesCopy<>mmToPulses THEN
				pulsesJogSpeedDesired:=JogSpeedDesired*mmToPulses;
				JogSpeedDesiredCopy:=JogSpeedDesired;
			END_IF;

		CALC_SPEED_PULSES:
			IF SpeedDesired<>SpeedDesiredCopy OR mmToPulsesCopy<>mmToPulses THEN
				pulsesSpeedDesired:=SpeedDesired*mmToPulses;
				SpeedDesiredCopy:=SpeedDesired;
			END_IF;

		CALC_ACC_PULSES:
			IF AccelerationDesired<>AccelerationDesiredCopy OR mmToPulsesCopy<>mmToPulses THEN
				pulsesAccelerationDesired:=AccelerationDesired*mmToPulses;
				AccelerationDesiredCopy:=AccelerationDesired;
			END_IF;

		CALC_ACC_MM:
			IF PulsesAccelerationDevice<>pulsesAccelerationDeviceCopy OR mmToPulsesCopy<>mmToPulses THEN
				mmAcceleration:=PulsesAccelerationDevice/mmToPulses;
				pulsesAccelerationDeviceCopy:=PulsesAccelerationDevice;
			END_IF

		CALC_DEC_PULSES:
			IF DecelerationDesired<>DecelerationDesiredCopy OR mmToPulsesCopy<>mmToPulses THEN
				pulsesDecelerationDesired:=DecelerationDesired*mmToPulses;
				DecelerationDesiredCopy:=DecelerationDesired;
			END_IF;

		CALC_DEC_MM:
			IF PulsesDecelerationDevice<>pulsesDecelerationDeviceCopy OR mmToPulsesCopy<>mmToPulses THEN
				mmDeceleration:=PulsesDecelerationDevice/mmToPulses;
				pulsesDecelerationDeviceCopy:=PulsesDecelerationDevice;
			END_IF

		CALC_SPEED_MMIN_PULSES:
			IF SpeedMminDesired<>SpeedMminDesiredCopy OR mmToPulsesCopy<>mmToPulses THEN
				pulsesSpeedDesired:=SpeedMminDesired*mmToPulses*1000/60; //Converting m/min to mm/s
				SpeedDesiredCopy:=SpeedDesired;
			END_IF;

		CALC_SPEED_MMIN:
			IF PulsesSpeedDevice<>pulsesSpeedDeviceCopy OR mmToPulsesCopy<>mmToPulses THEN
				SpeedMminDevice :=PulsesSpeedDevice*60/1000/mmToPulses;
				pulsesSpeedDeviceCopy:=PulsesSpeedDevice;
			END_IF;

		CALC_SPEED_MM:
			IF PulsesSpeedDevice<>pulsesSpeedDeviceCopy OR mmToPulsesCopy<>mmToPulses THEN
				SpeedDevice :=PulsesSpeedDevice/mmToPulses;
				pulsesSpeedDeviceCopy:=PulsesSpeedDevice;
			END_IF;

		CALC_SPEED_REVMIN_MMIN:
			IF RevMinSpeedDevice<>RevMinSpeedDeviceCopy OR mmToPulsesCopy<>mmToPulses THEN
				SpeedRpmToMmin :=RevMinSpeedDevice/mmToTurn/1000; //1000 to convert mm in meters
				RevMinSpeedDeviceCopy:=RevMinSpeedDevice;
			END_IF

	END_CASE

	TransDataCopy:=TransmissionData;
	mmToPulsesCopy:=mmToPulses;

END_FUNCTION_BLOCK
```

#### GetCalcVelocity.st
```iecst
(* TODO: Add your comment here *)
FUNCTION_BLOCK GetCalcVelocity

(* Escribe la velocidad en RPM en la variable interna *)
	IF xEn THEN
		IF xValid THEN
			rValor:=ABS(DINT_TO_REAL(diVelocidad_RPM));
		END_IF;
	ELSE
		rValor:=0.0;
	END_IF;

	(* Convierte de UM/Seg a M/MIN *)
	rm_rpm:= (((UINT_TO_REAL(uiEje)/10.0) / (UINT_TO_REAL(uiReductor))));
	iVel_lin:=REAL_TO_UINT((((rValor/1000) * rm_rpm)/1000)*600);

END_FUNCTION_BLOCK
```

#### MotorSpeedCalculation.st
```iecst
// It sets speed motor when enable is true otherewise SpeedMotor is Zero
FUNCTION_BLOCK MotorSpeedCalculation

	xChange := FALSE;

	// Enable function
	IF xEnable THEN
		// Conversion from mm/MIN a UM/seg
		m_rpm:= (((UINT_TO_REAL(uiRolllerPerimeter)/10.0)/ (UINT_TO_REAL(uiReductor)))); //	(mm/rev)
		rSpeedMotor := (((INT_TO_REAL((iSpSpeed))/60)/m_rpm) * 100 * rUnitsAtTheLoad ); //  (cm/seg : mm/rev)*100== (rev/seg)*1000000 == UM/seg
		IF xPrinterDirection = TRUE THEN
			rSpeedMotor:=-rSpeedMotor;
		END_IF;
	ELSE
		rSpeedMotor := 0;
	END_IF;
	// Trigger if change SP
	IF xChange = FALSE THEN
		IF Aux <> rSpeedMotor THEN
			xChange := TRUE;
			Aux := rSpeedMotor;
		END_IF;
	ELSE
	END_IF;

END_FUNCTION_BLOCK
```

#### SetCalcVelocity.st
```iecst
(* TODO: Add your comment here *)
FUNCTION_BLOCK SetCalcVelocity

	xChange:= FALSE;
	IF xEnMov THEN
		rSpeedInUnits := rSpeed / Mmin_TO_DriveUnitsRatio(rDiameter:=rAxisDiamter, rGearBox:=rReduction, rUnitsPerTurn:=rUnitsAtTheLoad);
	END_IF;

	// Trigger if change SP to a different value. Remove the activation of xChange when removing xEnMov input signal
	IF rSpeedInUnits <> rLastSpeedInUnits OR EDGEPOS(xEnMov) THEN
		xChange:= TRUE;
		rLastSpeedInUnits:=rSpeedInUnits;
	END_IF;

END_FUNCTION_BLOCK
```

### Program Logical/ExtPack/EFILib/EFILib_v1/Functions

#### ComandBoolEdge.st
```iecst
(* TODO: Add your comment here *)
FUNCTION ComandBoolEdge0

	IF Com = 0 OR Com = -1 THEN
		In := FALSE;
	END_IF

	IF Com = 1 THEN
		In := TRUE;
	END_IF

	Com := -1;
	ComandBoolEdge0 := In;

END_FUNCTION
```

#### DintTransfer.st
```iecst
(* TODO: Add your comment here *)
FUNCTION DintTransfer

// Out1
	LSint.0:=In.0;
	LSint.1:=In.1;
	LSint.2:=In.2;
	LSint.3:=In.3;
	LSint.4:=In.4;
	LSint.5:=In.5;
	LSint.6:=In.6;
	LSint.7:=In.7;
	LSint.8:=In.8;
	LSint.9:=In.9;
	LSint.10:=In.10;
	LSint.11:=In.11;
	LSint.12:=In.12;
	LSint.13:=In.13;
	LSint.14:=In.14;
	LSint.15:=In.15;

// Out2
	MSint.0:=In.16;
	MSint.1:=In.17;
	MSint.2:=In.18;
	MSint.3:=In.19;
	MSint.4:=In.20;
	MSint.5:=In.21;
	MSint.6:=In.22;
	MSint.7:=In.23;
	MSint.8:=In.24;
	MSint.9:=In.25;
	MSint.10:=In.26;
	MSint.11:=In.27;
	MSint.12:=In.28;
	MSint.13:=In.29;
	MSint.14:=In.30;
	MSint.15:=In.31;

	DintTransfer := TRUE;

END_FUNCTION
```

#### Mmin_TO_DriveUnitsRatio.st
```iecst
(* TODO: Add your comment here *)
FUNCTION Mmin_TO_DriveUnitsRatio

	//Protection of values to avoid infinite values
	rDiameter := MAX(rDiameter, 10);
	IF rGearBox = 0 THEN rGearBox:=1; END_IF

	Mmin_TO_DriveUnitsRatio:=(60 * rDiameter) / (1000 * rGearBox * rUnitsPerTurn);

END_FUNCTION
```

#### PLC.st
```iecst
(* Load initial script for PLC. VOID *)
FUNCTION PLC_Init

	//PLC String name creation
	plcStruct.sVersion := 'PLC v';
	brsitoa(plcStruct.iVersion0, ADR(strAux));
	brsstrcat(ADR(plcStruct.sVersion), ADR(strAux));
	strAux := '.';
	brsstrcat(ADR(plcStruct.sVersion), ADR(strAux));
	brsitoa(plcStruct.iVersion1, ADR(strAux));
	brsstrcat(ADR(plcStruct.sVersion), ADR(strAux));
	strAux := '.';
	brsstrcat(ADR(plcStruct.sVersion), ADR(strAux));
	brsitoa(plcStruct.iVersion2, ADR(strAux));
	brsstrcat(ADR(plcStruct.sVersion), ADR(strAux));
	strAux := '.';
	brsstrcat(ADR(plcStruct.sVersion), ADR(strAux));
	brsitoa(plcStruct.iVersion3, ADR(strAux));
	brsstrcat(ADR(plcStruct.sVersion), ADR(strAux));

	PLC_Init := TRUE;

END_FUNCTION
```

#### StatusTemperatureInput.st
```iecst
// Temperature Input state
FUNCTION StatusTemperatureInput

	//If Module is NOT OK, directly It returns an alarm, Block.Al.xModuleTemp0X

	//Channels iInputTemperatureNumber from 1 to 4 in iStatusInputTemp01
	iStatusTemperatureInput:= SHR(iStatusTempInput01,(iTemperatureInputNumber-1)*2) AND 16#03;
	// Ouput bolean, value 3 means that there is an opencircuit in PT100
	IF iStatusTemperatureInput > 2 THEN
		StatusTemperatureInput:= TRUE;
	ELSE
		StatusTemperatureInput:= FALSE;
	END_IF

END_FUNCTION
```

#### Time.st
```iecst
(* Time in ms to run a distance in mm with speed in m/min. TIME *)
FUNCTION TimeFromMmAndMmin

	IF rSpeed = 0 THEN
		TimeFromMmAndMmin := T#24d; //Value close to the maximum
	END_IF

	TimeFromMmAndMmin := REAL_TO_TIME(rDistance * 60 / rSpeed);

END_FUNCTION
```

#### UDINTFromComms.st
```iecst
(* Assignation of a UDINT Double value from an array *)
FUNCTION UDINTFromComms
//	indexLSB	UINT	FALSE	VAR_INPUT					 	 	 	 	69
//	comsArray	INT[0..9999]	TRUE	VAR_INPUT					 	 	 	 	70
	UDINTFromComms := INT_TO_UINT(comsArray[indexLSB]) + 16#10000 * INT_TO_UINT(comsArray[indexLSB+1]);
END_FUNCTION
```

#### UDINTToComms.st
```iecst
(* Insert a UDINT value in an array for comms *)
FUNCTION UDINTToComms

	//	value	UDINT	FALSE	VAR_INPUT
	//	indexLSB	UINT	FALSE	VAR_INPUT
	//	comsArray	INT[0..9999]	TRUE	VAR_INPUT

	comsArray[indexLSB] :=	UDINT_TO_INT(value AND 16#0000FFFF);
	comsArray[indexLSB+1] :=UDINT_TO_INT(SHR(value AND 16#FFFF0000,16));

	UDINTToComms:=TRUE;

END_FUNCTION
```

#### UINT_SUB.st
```iecst
(* TODO: Add your comment here *)
FUNCTION UINT_SUB

	//Protection of values to avoid infinite values
	IF Minuend >= Subtrahend THEN
		UINT_SUB := Minuend - Subtrahend;
	ELSE
		UINT_SUB := 0;
	END_IF

END_FUNCTION
```

### Inks.var
```iecst
VAR
	gIndexInks : UINT := 0;
END_VAR
```

- ActTempToPID.xlsx (binary file, 22563 bytes)
- InkHeaterTankProcess.graphml (not shown)

- InkHeaterTankSystem.graphml (not shown)

- InksControl.graphml (not shown)

- PrimingSystemProcess.graphml (not shown)

- TemperatureOut.mm (not shown)

### Program Logical/ExtPack/InksCtrl/InksCtrl_v3/InitInksCtrl (IEC)

#### InitInksCtrl.st - Init Inks Control
```iecst
PROGRAM _CYCLIC
	gIndexInks := 1;
END_PROGRAM
```

### Program Logical/ExtPack/InksCtrl/InksCtrl_v3/InksCtrl (IEC)

#### safetyPre.st - Safet preconversions
```iecst
ACTION safetyPre:

//	//Limits of the analog control signal are 0V and 5V
//	IF parBar.rLowPumpLimitNeg < 0 	THEN parBar.rLowPumpLimitNeg := 0; END_IF
//	IF parBar.rLowPumpLimitPos < 0 	THEN parBar.rLowPumpLimitPos := 0; END_IF
//	IF parBar.rHighPumpLimitNeg > 5 	THEN parBar.rHighPumpLimitNeg := 5; END_IF
//	IF parBar.rHighPumpLimitPos > 5 	THEN parBar.rHighPumpLimitPos := 5; END_IF
//
//	//If the Max value is too low, we assign the minimum value
//	IF parBar.rHighPumpLimitNeg < gc_rMinDiffMinMaxCtrlVoltage THEN parBar.rHighPumpLimitNeg := gc_rMinDiffMinMaxCtrlVoltage; END_IF
//	IF parBar.rHighPumpLimitPos < gc_rMinDiffMinMaxCtrlVoltage THEN parBar.rHighPumpLimitPos := gc_rMinDiffMinMaxCtrlVoltage; END_IF
//
	inks.parameters.Temp.iBarsWithSameBlock:=MAX(inks.parameters.Temp.iBarsWithSameBlock,1);

END_ACTION
```

#### conversionsPre.st - Preconversions
```iecst
ACTION conversionsPre:

	//Individual DripTime of the bar
	tiDripTime:= MIN(inks.parSw.tiDripTime, INKS_DRIP_TIME_MAX);

	//Maximum DripTime of all the "brother" bars. And to be sure DripTimeMax is not smaller than DripTime
	tiDripTimeMax:= MAX( MIN(inks.parameters.tiDripTimeMax, INKS_DRIP_TIME_MAX), tiDripTime);

	//Level
	IF parBar.xTypeTankSensorAnalog THEN
		//tests level sensor.
		fbFilterLevelSensor(Enable:=TRUE,
							In:=(((INT_TO_REAL(inks.signals.in.iInTankLevel-16383)*1500)/16384.0)),
							WindowLength:=60);

		rTankLevelmm:= fbFilterLevelSensor.Out;

		rTankLevelPercent:= LIMIT(0, (rTankLevelmm/2.35), 100);

	END_IF

	//filters
	inks.status.Temp.rTemp:= INT_TO_REAL(inks.signals.in.iTemperatureRaw)/10.0;
	inks.status.Temp.rTempTank:= INT_TO_REAL(inks.signals.in.iTemperatureTankRaw)/10.0;

	//Vacuum gauge inputs
	//
	//4-20mA Input Current loop
	// iVacuumXRaw: It is an integer value from 0 to 32767.
	// It is configured in current loop, 4mA is assigned TO 6553,
	// lower than 1000 are reported as 0 by GUI
	// and lower than -8000 are reported as pressure gauge disconnected
	// Checked with M4

	//
	// fbFilterMovingPressure1
	//	iSamplesVacuum1: 60 samples
	IF inks.signals.in.iVacuum1Raw > 1000 THEN
		rInputFilterVacuum1:= ((INT_TO_REAL(inks.signals.in.iVacuum1Raw)* inks.parameters.parBar.rVacuumSensorSpan)/32767.0)+inks.parameters.parBar.rVacuumSensorOffset;
		fbFilterMovingPressure1(Enable:=TRUE ,
			In:=rInputFilterVacuum1,
			WindowLength:=iSamplesVacuum1 ,
			);
		rVacuum1B:= fbFilterMovingPressure1.Out;

	ELSE
		rVacuum1B:=0;
		//When simulators or printheads are not installed, this value is reported to GUI
		//For that, GUI shows zeros because PLC vaues lower than 1000
		// xAlrVacuum1 has to be activated
	END_IF

	// Filter average of the input pressure sensor
	(*La entrada tiene valores de 0 a 32767, los 4mA corresponden a 6553*)
	IF inks.signals.in.iVacuum2Raw > 1000 THEN
		rInputFilterVacuum2:= ((INT_TO_REAL(inks.signals.in.iVacuum2Raw)* inks.parameters.parBar.rVacuumSensorSpan)/32767.0)+inks.parameters.parBar.rVacuumSensorOffset;
		fbFilterMovingPressure2(
			Enable:=TRUE ,
			In:=rInputFilterVacuum2,
			WindowLength:=iSamplesVacuum2 ,
			);
		rVacuum2B:= fbFilterMovingPressure2.Out;

	ELSE
		rVacuum2B:=0;
		//When simulators or printheads are not installed, this value is reported to GUI
		//For that, GUI shows zeros because PLC values lower than 1000
		// xAlrVacuum2 has to be activated
	END_IF

	//Assign vacuum data to status for external viewing
	inks.status.rVacuum1 := rVacuum1B;
	inks.status.rVacuum2 := rVacuum2B;

	////Out DC Pumps treatment SetPoints
	rLowPumpLimitNeg 	:=parBar.rLowPumpLimitNeg;
	rHighPumpLimitNeg 	:=parBar.rHighPumpLimitNeg;
	IF (rHighPumpLimitNeg - rLowPumpLimitNeg) < Ic_rMinDiffMinMaxCtrlVoltage THEN
		rLowPumpLimitNeg 	:=parBar.rHighPumpLimitNeg - Ic_rMinDiffMinMaxCtrlVoltage;
	END_IF
	rSlopePumpNeg 		:=(rHighPumpLimitNeg-rLowPumpLimitNeg)/100;

	rLowPumpLimitPos 	:=parBar.rLowPumpLimitPos;
	rHighPumpLimitPos 	:=parBar.rHighPumpLimitPos;
	IF (rHighPumpLimitPos - rLowPumpLimitPos) < Ic_rMinDiffMinMaxCtrlVoltage THEN
		rLowPumpLimitPos 	:=parBar.rHighPumpLimitPos - Ic_rMinDiffMinMaxCtrlVoltage;
	END_IF
	rSlopePumpPos 		:=(rHighPumpLimitPos-rLowPumpLimitPos)/100;

	// Bar number installed in block from Mapping
	iBarNumberInBlock := (inks.parSw.Config.iMappingBar -1) MOD inks.parameters.Temp.iBarsWithSameBlock;

	rVacuumSensorMax := inks.parameters.parBar.rVacuumSensorSpan + inks.parameters.parBar.rVacuumSensorOffset;

END_ACTION
```
